% RSLogix 500 project TEST DENHAM_BAK006.RSS, saved by version 11.00.00.00 %
PROJECT "UNTITLED"    % processor: MicroLogix 1400 %

PROGRAM FILES
  LAD 2   184 rungs

DATA FILES
  O0 OUTPUT  8 elements
  I1 INPUT  17 elements
  S2 STATUS  66 elements
  B3 BINARY  6 elements
  T4 TIMER  28 elements
  C5 COUNTER  1 elements
  R6 CONTROL  1 elements
  N7 INTEGER  41 elements
  F8 FLOAT  8 elements
  PD11   2 elements

LADDER 2
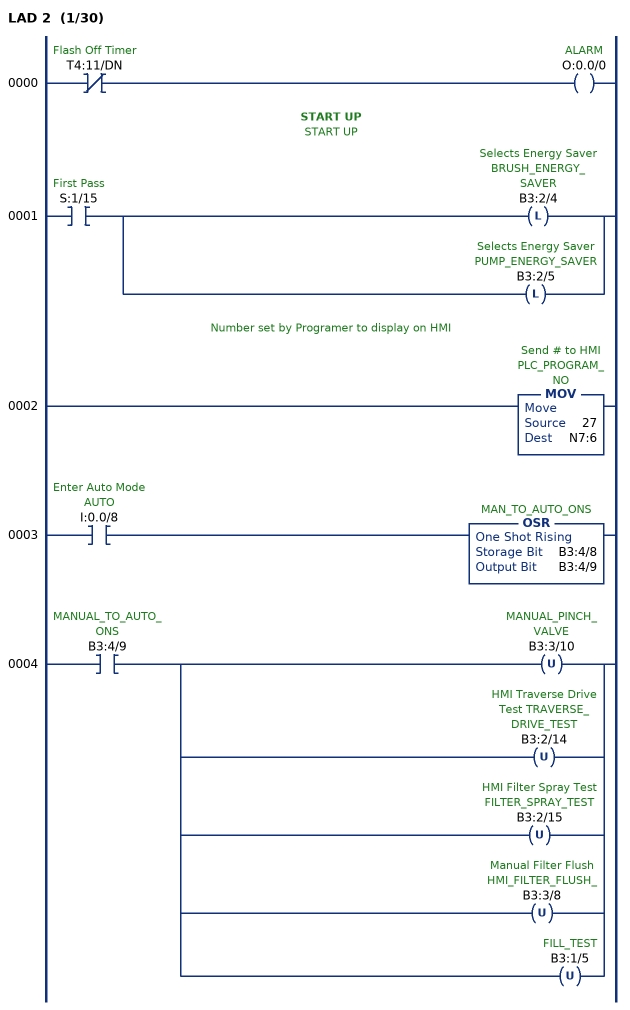
% Rung: 0 %
SOR XIO T4:11/DN OTE O:0.0/0 EOR
%   T4:11  "Flash Off Timer" %
%   O:0.0/0  ALARM %
% Rung: 1 %
% TITLE: START UP %
% START UP %
SOR XIC S:1/15 BST OTL B3:2/4 NXB OTL B3:2/5 BND EOR
%   S:1/15  "First Pass" %
%   B3:2/4  BRUSH_ENERGY_SAVER  "Selects Energy Saver" %
%   B3:2/5  PUMP_ENERGY_SAVER  "Selects Energy Saver" %
% Rung: 2 %
% Number set by Programer to display on HMI %
SOR MOV 27 N7:6 EOR
%   N7:6  PLC_PROGRAM_NO  "Send # to HMI" %
% Rung: 3 %
SOR XIC I:0.0/8 OSR B3:4/8 B3:4/9 EOR
%   I:0.0/8  AUTO  "Enter Auto Mode" %
%   B3:4/8  MAN_TO_AUTO_ONS %
%   B3:4/9  MANUAL_TO_AUTO_ONS %
% Rung: 4 %
SOR XIC B3:4/9 BST OTU B3:3/10 NXB BST OTU B3:2/14 NXB BST OTU B3:2/15 NXB BST OTU B3:3/8 NXB OTU B3:1/5 BND BND BND BND EOR
%   B3:4/9  MANUAL_TO_AUTO_ONS %
%   B3:3/10  MANUAL_PINCH_VALVE %
%   B3:2/14  TRAVERSE_DRIVE_TEST  "HMI Traverse Drive Test" %
%   B3:2/15  FILTER_SPRAY_TEST  "HMI Filter Spray Test" %
%   B3:3/8  HMI_FILTER_FLUSH_  "Manual Filter Flush" %
%   B3:1/5  FILL_TEST %

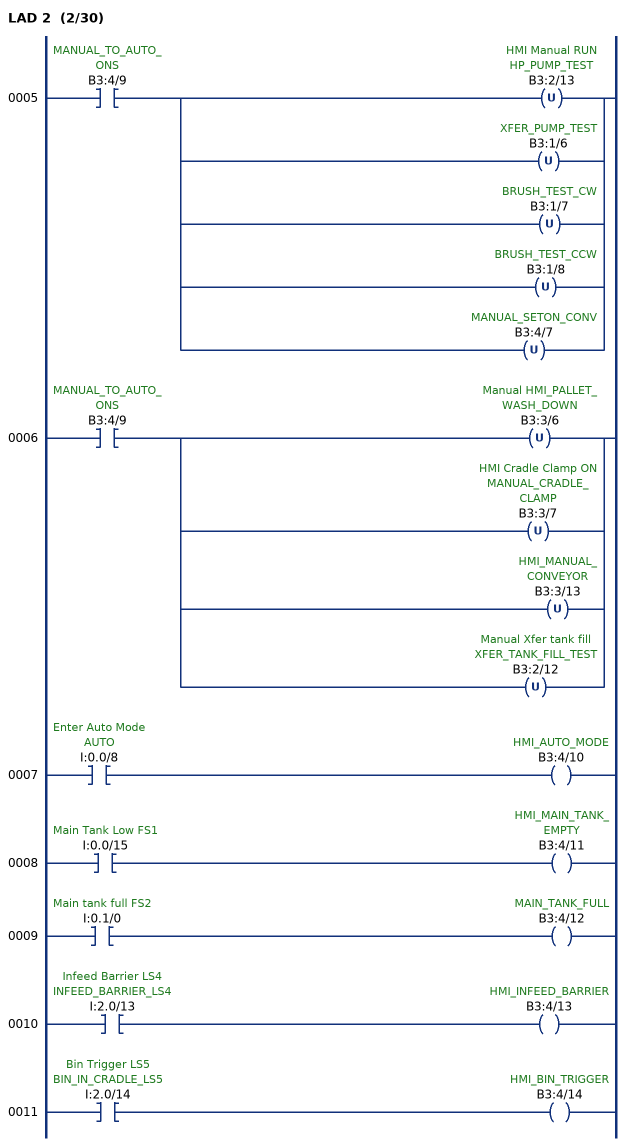
% Rung: 5 %
SOR XIC B3:4/9 BST OTU B3:2/13 NXB BST OTU B3:1/6 NXB BST OTU B3:1/7 NXB BST OTU B3:1/8 NXB OTU B3:4/7 BND BND BND BND EOR
%   B3:4/9  MANUAL_TO_AUTO_ONS %
%   B3:2/13  HP_PUMP_TEST  "HMI Manual RUN" %
%   B3:1/6  XFER_PUMP_TEST %
%   B3:1/7  BRUSH_TEST_CW %
%   B3:1/8  BRUSH_TEST_CCW %
%   B3:4/7  MANUAL_SETON_CONV %
% Rung: 6 %
SOR XIC B3:4/9 BST OTU B3:3/6 NXB BST OTU B3:3/7 NXB BST OTU B3:3/13 NXB OTU B3:2/12 BND BND BND EOR
%   B3:4/9  MANUAL_TO_AUTO_ONS %
%   B3:3/6  HMI_PALLET_WASH_DOWN  "Manual" %
%   B3:3/7  MANUAL_CRADLE_CLAMP  "HMI Cradle Clamp ON" %
%   B3:3/13  HMI_MANUAL_CONVEYOR %
%   B3:2/12  XFER_TANK_FILL_TEST  "Manual Xfer tank fill" %
% Rung: 7 %
SOR XIC I:0.0/8 OTE B3:4/10 EOR
%   I:0.0/8  AUTO  "Enter Auto Mode" %
%   B3:4/10  HMI_AUTO_MODE %
% Rung: 8 %
SOR XIC I:0.0/15 OTE B3:4/11 EOR
%   I:0.0/15  FS1  "Main Tank Low" %
%   B3:4/11  HMI_MAIN_TANK_EMPTY %
% Rung: 9 %
SOR XIC I:0.1/0 OTE B3:4/12 EOR
%   I:0.1/0  FS2  "Main tank full" %
%   B3:4/12  MAIN_TANK_FULL %
% Rung: 10 %
SOR XIC I:2.0/13 OTE B3:4/13 EOR
%   I:2.0/13  INFEED_BARRIER_LS4  "Infeed Barrier LS4" %
%   B3:4/13  HMI_INFEED_BARRIER %
% Rung: 11 %
SOR XIC I:2.0/14 OTE B3:4/14 EOR
%   I:2.0/14  BIN_IN_CRADLE_LS5  "Bin Trigger LS5" %
%   B3:4/14  HMI_BIN_TRIGGER %

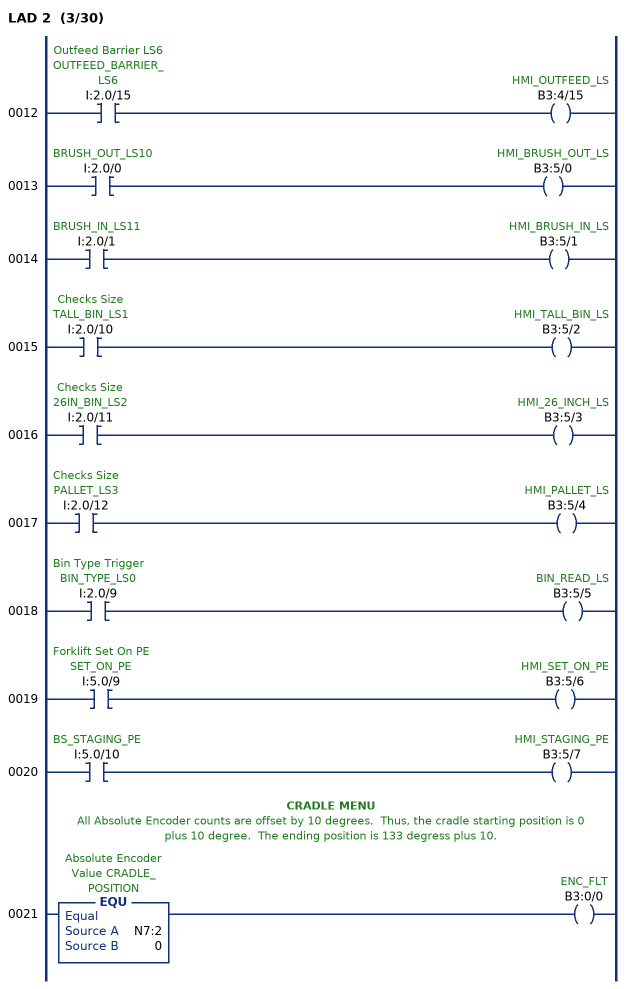
% Rung: 12 %
SOR XIC I:2.0/15 OTE B3:4/15 EOR
%   I:2.0/15  OUTFEED_BARRIER_LS6  "Outfeed Barrier LS6" %
%   B3:4/15  HMI_OUTFEED_LS %
% Rung: 13 %
SOR XIC I:2.0/0 OTE B3:5/0 EOR
%   I:2.0/0  BRUSH_OUT_LS10 %
%   B3:5/0  HMI_BRUSH_OUT_LS %
% Rung: 14 %
SOR XIC I:2.0/1 OTE B3:5/1 EOR
%   I:2.0/1  BRUSH_IN_LS11 %
%   B3:5/1  HMI_BRUSH_IN_LS %
% Rung: 15 %
SOR XIC I:2.0/10 OTE B3:5/2 EOR
%   I:2.0/10  TALL_BIN_LS1  "Checks Size" %
%   B3:5/2  HMI_TALL_BIN_LS %
% Rung: 16 %
SOR XIC I:2.0/11 OTE B3:5/3 EOR
%   I:2.0/11  26IN_BIN_LS2  "Checks Size" %
%   B3:5/3  HMI_26_INCH_LS %
% Rung: 17 %
SOR XIC I:2.0/12 OTE B3:5/4 EOR
%   I:2.0/12  PALLET_LS3  "Checks Size" %
%   B3:5/4  HMI_PALLET_LS %
% Rung: 18 %
SOR XIC I:2.0/9 OTE B3:5/5 EOR
%   I:2.0/9  BIN_TYPE_LS0  "Bin Type Trigger" %
%   B3:5/5  BIN_READ_LS %
% Rung: 19 %
SOR XIC I:5.0/9 OTE B3:5/6 EOR
%   I:5.0/9  SET_ON_PE  "Forklift Set On PE" %
%   B3:5/6  HMI_SET_ON_PE %
% Rung: 20 %
SOR XIC I:5.0/10 OTE B3:5/7 EOR
%   I:5.0/10  BS_STAGING_PE %
%   B3:5/7  HMI_STAGING_PE %
% Rung: 21 %
% TITLE: CRADLE MENU %
% All Absolute Encoder counts are offset by 10 degrees.  Thus, the cradle starting position is 0 plus 10 degree.  The ending position is 133 degress plus 10. %
SOR EQU N7:2 0 OTE B3:0/0 EOR
%   N7:2  CRADLE_POSITION  "Absolute Encoder Value" %
%   B3:0/0  ENC_FLT %

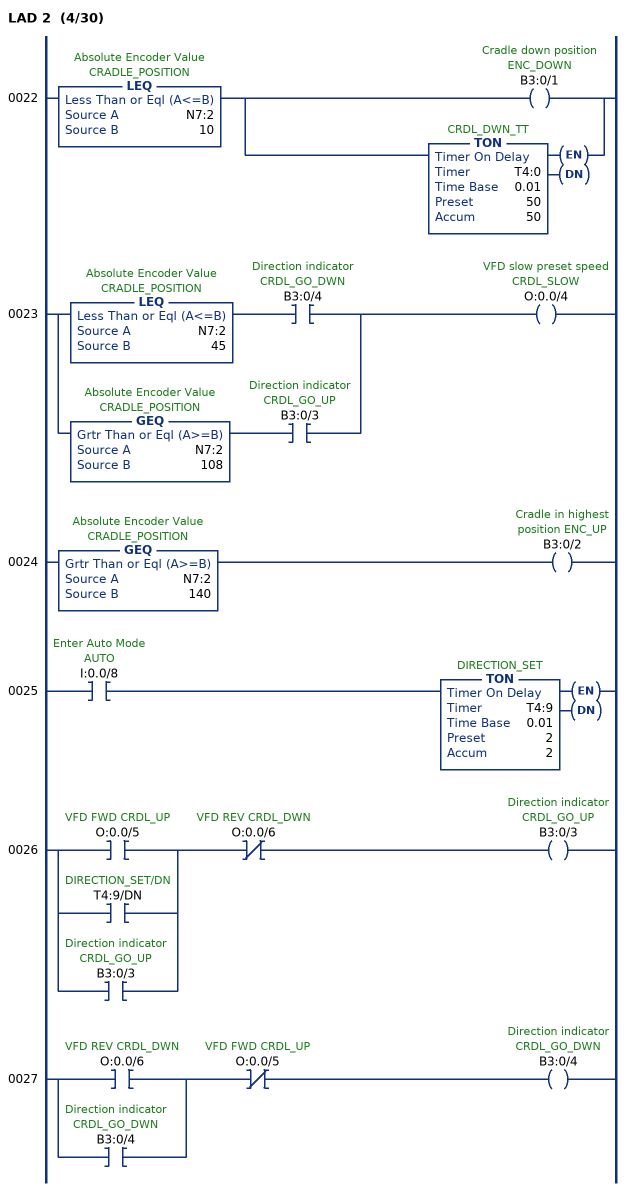
% Rung: 22 %
SOR LEQ N7:2 10 BST OTE B3:0/1 NXB TON T4:0 0.01 50 50 BND EOR
%   N7:2  CRADLE_POSITION  "Absolute Encoder Value" %
%   B3:0/1  ENC_DOWN  "Cradle down position" %
%   T4:0  CRDL_DWN_TT %
% Rung: 23 %
SOR BST LEQ N7:2 45 XIC B3:0/4 NXB GEQ N7:2 108 XIC B3:0/3 BND OTE O:0.0/4 EOR
%   N7:2  CRADLE_POSITION  "Absolute Encoder Value" %
%   B3:0/4  CRDL_GO_DWN  "Direction indicator" %
%   B3:0/3  CRDL_GO_UP  "Direction indicator" %
%   O:0.0/4  CRDL_SLOW  "VFD slow preset speed" %
% Rung: 24 %
SOR GEQ N7:2 140 OTE B3:0/2 EOR
%   N7:2  CRADLE_POSITION  "Absolute Encoder Value" %
%   B3:0/2  ENC_UP  "Cradle in highest position" %
% Rung: 25 %
SOR XIC I:0.0/8 TON T4:9 0.01 2 2 EOR
%   I:0.0/8  AUTO  "Enter Auto Mode" %
%   T4:9  DIRECTION_SET %
% Rung: 26 %
SOR BST XIC O:0.0/5 NXB XIC T4:9/DN NXB XIC B3:0/3 BND XIO O:0.0/6 OTE B3:0/3 EOR
%   O:0.0/5  CRDL_UP  "VFD FWD" %
%   T4:9  DIRECTION_SET %
%   B3:0/3  CRDL_GO_UP  "Direction indicator" %
%   O:0.0/6  CRDL_DWN  "VFD REV" %
% Rung: 27 %
SOR BST XIC O:0.0/6 NXB XIC B3:0/4 BND XIO O:0.0/5 OTE B3:0/4 EOR
%   O:0.0/6  CRDL_DWN  "VFD REV" %
%   B3:0/4  CRDL_GO_DWN  "Direction indicator" %
%   O:0.0/5  CRDL_UP  "VFD FWD" %

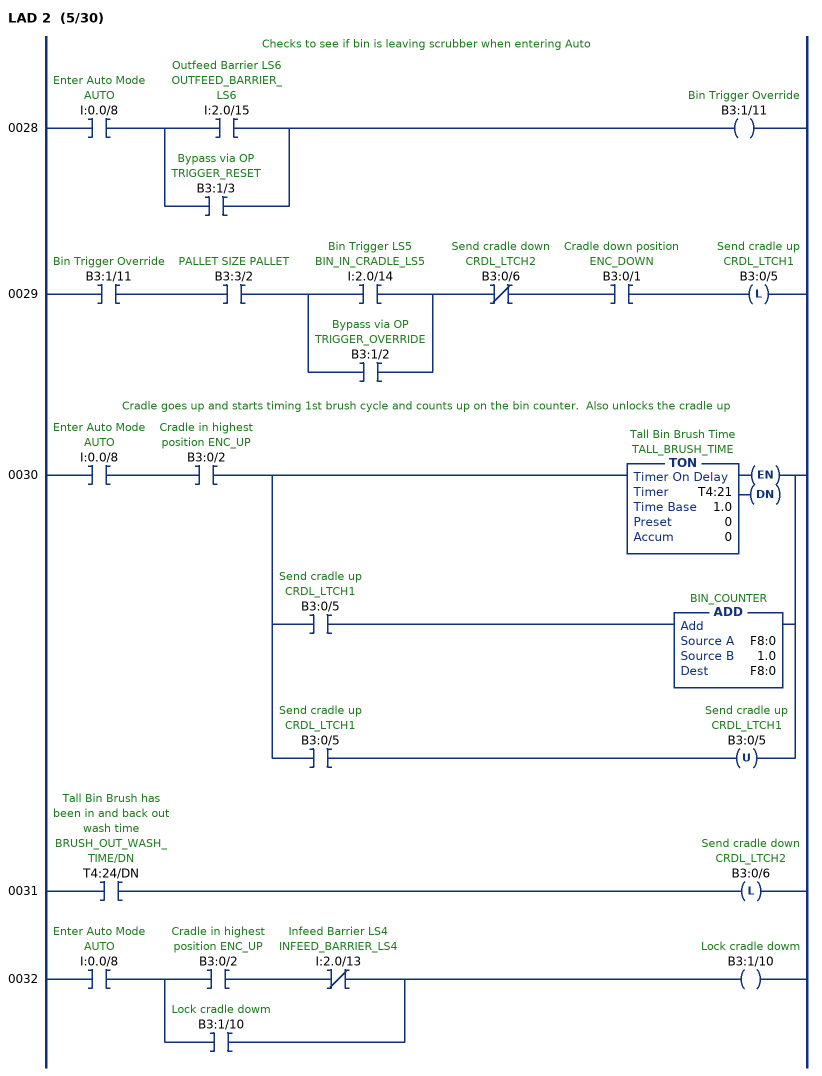
% Rung: 28 %
% Checks to see if bin is leaving scrubber when entering Auto %
SOR XIC I:0.0/8 BST XIC I:2.0/15 NXB XIC B3:1/3 BND OTE B3:1/11 EOR
%   I:0.0/8  AUTO  "Enter Auto Mode" %
%   I:2.0/15  OUTFEED_BARRIER_LS6  "Outfeed Barrier LS6" %
%   B3:1/3  TRIGGER_RESET  "Bypass via OP" %
%   B3:1/11  "Bin Trigger Override" %
% Rung: 29 %
SOR XIC B3:1/11 XIC B3:3/2 BST XIC I:2.0/14 NXB XIC B3:1/2 BND XIO B3:0/6 XIC B3:0/1 OTL B3:0/5 EOR
%   B3:1/11  "Bin Trigger Override" %
%   B3:3/2  PALLET  "PALLET SIZE" %
%   I:2.0/14  BIN_IN_CRADLE_LS5  "Bin Trigger LS5" %
%   B3:1/2  TRIGGER_OVERRIDE  "Bypass via OP" %
%   B3:0/6  CRDL_LTCH2  "Send cradle down" %
%   B3:0/1  ENC_DOWN  "Cradle down position" %
%   B3:0/5  CRDL_LTCH1  "Send cradle up" %
% Rung: 30 %
% Cradle goes up and starts timing 1st brush cycle and counts up on the bin counter.  Also unlocks the cradle up %
SOR XIC I:0.0/8 XIC B3:0/2 BST TON T4:21 1.0 0 0 NXB BST XIC B3:0/5 ADD F8:0 1.0 F8:0 NXB XIC B3:0/5 OTU B3:0/5 BND BND EOR
%   I:0.0/8  AUTO  "Enter Auto Mode" %
%   B3:0/2  ENC_UP  "Cradle in highest position" %
%   T4:21  TALL_BRUSH_TIME  "Tall Bin Brush Time" %
%   B3:0/5  CRDL_LTCH1  "Send cradle up" %
%   F8:0  BIN_COUNTER %
% Rung: 31 %
SOR XIC T4:24/DN OTL B3:0/6 EOR
%   T4:24  BRUSH_OUT_WASH_TIME  "Tall Bin Brush has been in and back out wash time" %
%   B3:0/6  CRDL_LTCH2  "Send cradle down" %
% Rung: 32 %
SOR XIC I:0.0/8 BST XIC B3:0/2 XIO I:2.0/13 NXB XIC B3:1/10 BND OTE B3:1/10 EOR
%   I:0.0/8  AUTO  "Enter Auto Mode" %
%   B3:0/2  ENC_UP  "Cradle in highest position" %
%   I:2.0/13  INFEED_BARRIER_LS4  "Infeed Barrier LS4" %
%   B3:1/10  "Lock cradle dowm" %

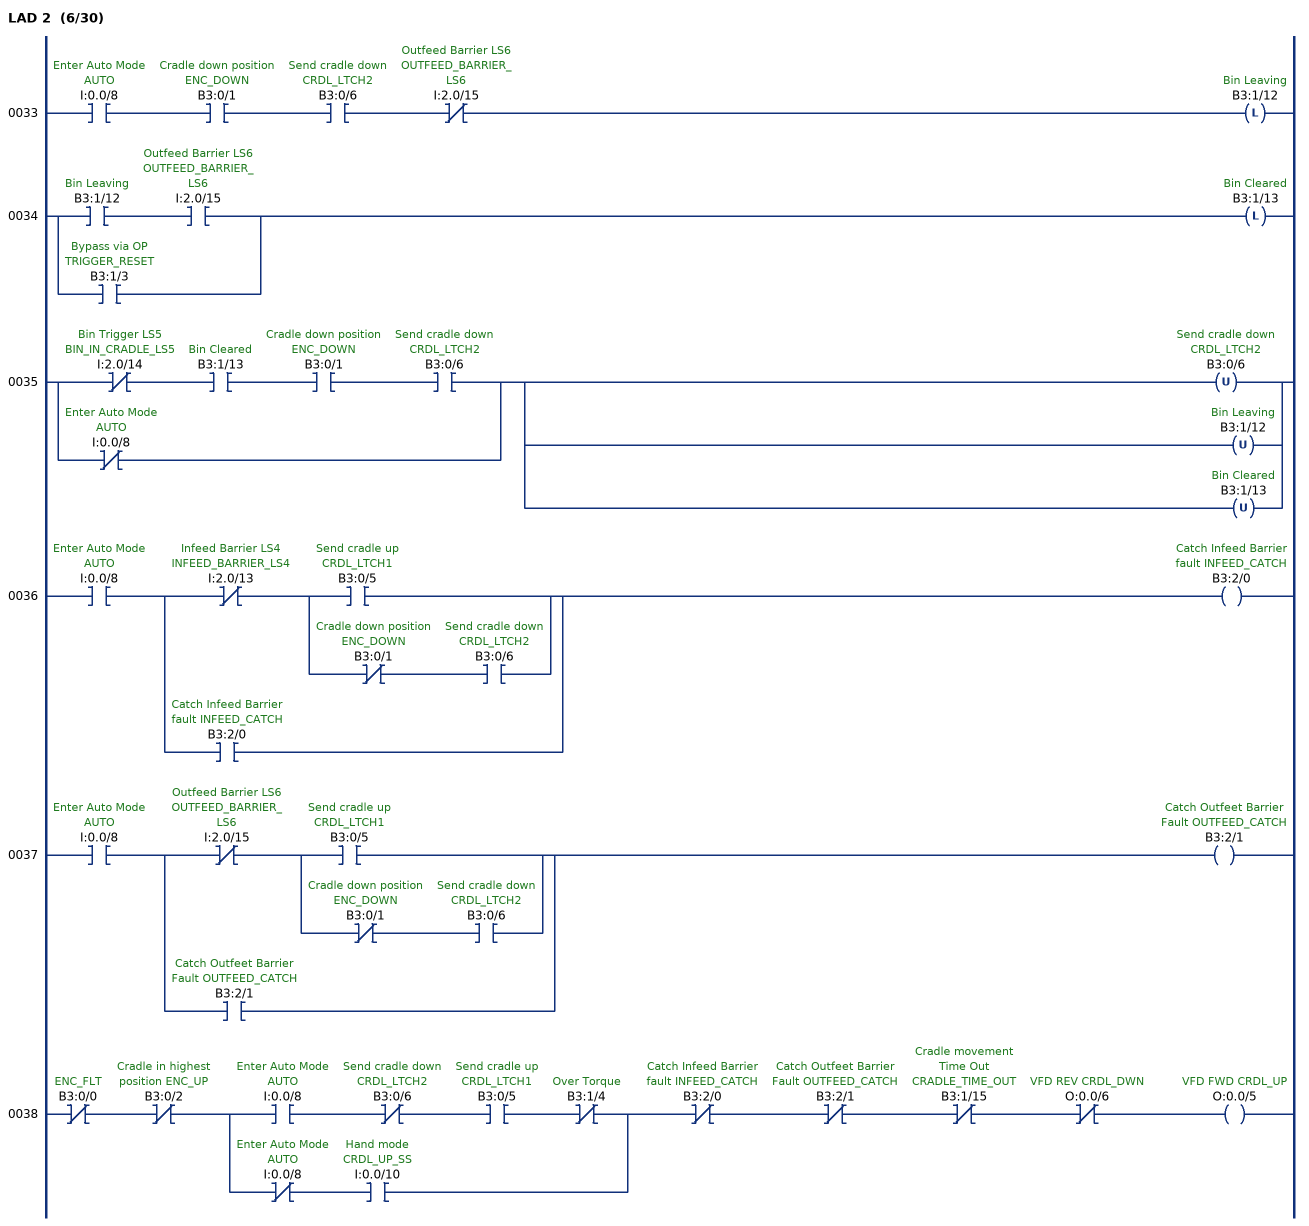
% Rung: 33 %
SOR XIC I:0.0/8 XIC B3:0/1 XIC B3:0/6 XIO I:2.0/15 OTL B3:1/12 EOR
%   I:0.0/8  AUTO  "Enter Auto Mode" %
%   B3:0/1  ENC_DOWN  "Cradle down position" %
%   B3:0/6  CRDL_LTCH2  "Send cradle down" %
%   I:2.0/15  OUTFEED_BARRIER_LS6  "Outfeed Barrier LS6" %
%   B3:1/12  "Bin Leaving" %
% Rung: 34 %
SOR BST XIC B3:1/12 XIC I:2.0/15 NXB XIC B3:1/3 BND OTL B3:1/13 EOR
%   B3:1/12  "Bin Leaving" %
%   I:2.0/15  OUTFEED_BARRIER_LS6  "Outfeed Barrier LS6" %
%   B3:1/3  TRIGGER_RESET  "Bypass via OP" %
%   B3:1/13  "Bin Cleared" %
% Rung: 35 %
SOR BST XIO I:2.0/14 XIC B3:1/13 XIC B3:0/1 XIC B3:0/6 NXB XIO I:0.0/8 BND BST OTU B3:0/6 NXB BST OTU B3:1/12 NXB OTU B3:1/13 BND BND EOR
%   I:2.0/14  BIN_IN_CRADLE_LS5  "Bin Trigger LS5" %
%   B3:1/13  "Bin Cleared" %
%   B3:0/1  ENC_DOWN  "Cradle down position" %
%   B3:0/6  CRDL_LTCH2  "Send cradle down" %
%   I:0.0/8  AUTO  "Enter Auto Mode" %
%   B3:1/12  "Bin Leaving" %
% Rung: 36 %
SOR XIC I:0.0/8 BST XIO I:2.0/13 BST XIC B3:0/5 NXB XIO B3:0/1 XIC B3:0/6 BND NXB XIC B3:2/0 BND OTE B3:2/0 EOR
%   I:0.0/8  AUTO  "Enter Auto Mode" %
%   I:2.0/13  INFEED_BARRIER_LS4  "Infeed Barrier LS4" %
%   B3:0/5  CRDL_LTCH1  "Send cradle up" %
%   B3:0/1  ENC_DOWN  "Cradle down position" %
%   B3:0/6  CRDL_LTCH2  "Send cradle down" %
%   B3:2/0  INFEED_CATCH  "Catch Infeed Barrier fault" %
% Rung: 37 %
SOR XIC I:0.0/8 BST XIO I:2.0/15 BST XIC B3:0/5 NXB XIO B3:0/1 XIC B3:0/6 BND NXB XIC B3:2/1 BND OTE B3:2/1 EOR
%   I:0.0/8  AUTO  "Enter Auto Mode" %
%   I:2.0/15  OUTFEED_BARRIER_LS6  "Outfeed Barrier LS6" %
%   B3:0/5  CRDL_LTCH1  "Send cradle up" %
%   B3:0/1  ENC_DOWN  "Cradle down position" %
%   B3:0/6  CRDL_LTCH2  "Send cradle down" %
%   B3:2/1  OUTFEED_CATCH  "Catch Outfeet Barrier Fault" %
% Rung: 38 %
SOR XIO B3:0/0 XIO B3:0/2 BST XIC I:0.0/8 XIO B3:0/6 XIC B3:0/5 XIO B3:1/4 NXB XIO I:0.0/8 XIC I:0.0/10 BND XIO B3:2/0 XIO B3:2/1 XIO B3:1/15 XIO O:0.0/6 OTE O:0.0/5 EOR
%   B3:0/0  ENC_FLT %
%   B3:0/2  ENC_UP  "Cradle in highest position" %
%   I:0.0/8  AUTO  "Enter Auto Mode" %
%   B3:0/6  CRDL_LTCH2  "Send cradle down" %
%   B3:0/5  CRDL_LTCH1  "Send cradle up" %
%   B3:1/4  "Over Torque" %
%   I:0.0/10  CRDL_UP_SS  "Hand mode" %
%   B3:2/0  INFEED_CATCH  "Catch Infeed Barrier fault" %
%   B3:2/1  OUTFEED_CATCH  "Catch Outfeet Barrier Fault" %
%   B3:1/15  CRADLE_TIME_OUT  "Cradle movement Time Out" %
%   O:0.0/6  CRDL_DWN  "VFD REV" %
%   O:0.0/5  CRDL_UP  "VFD FWD" %

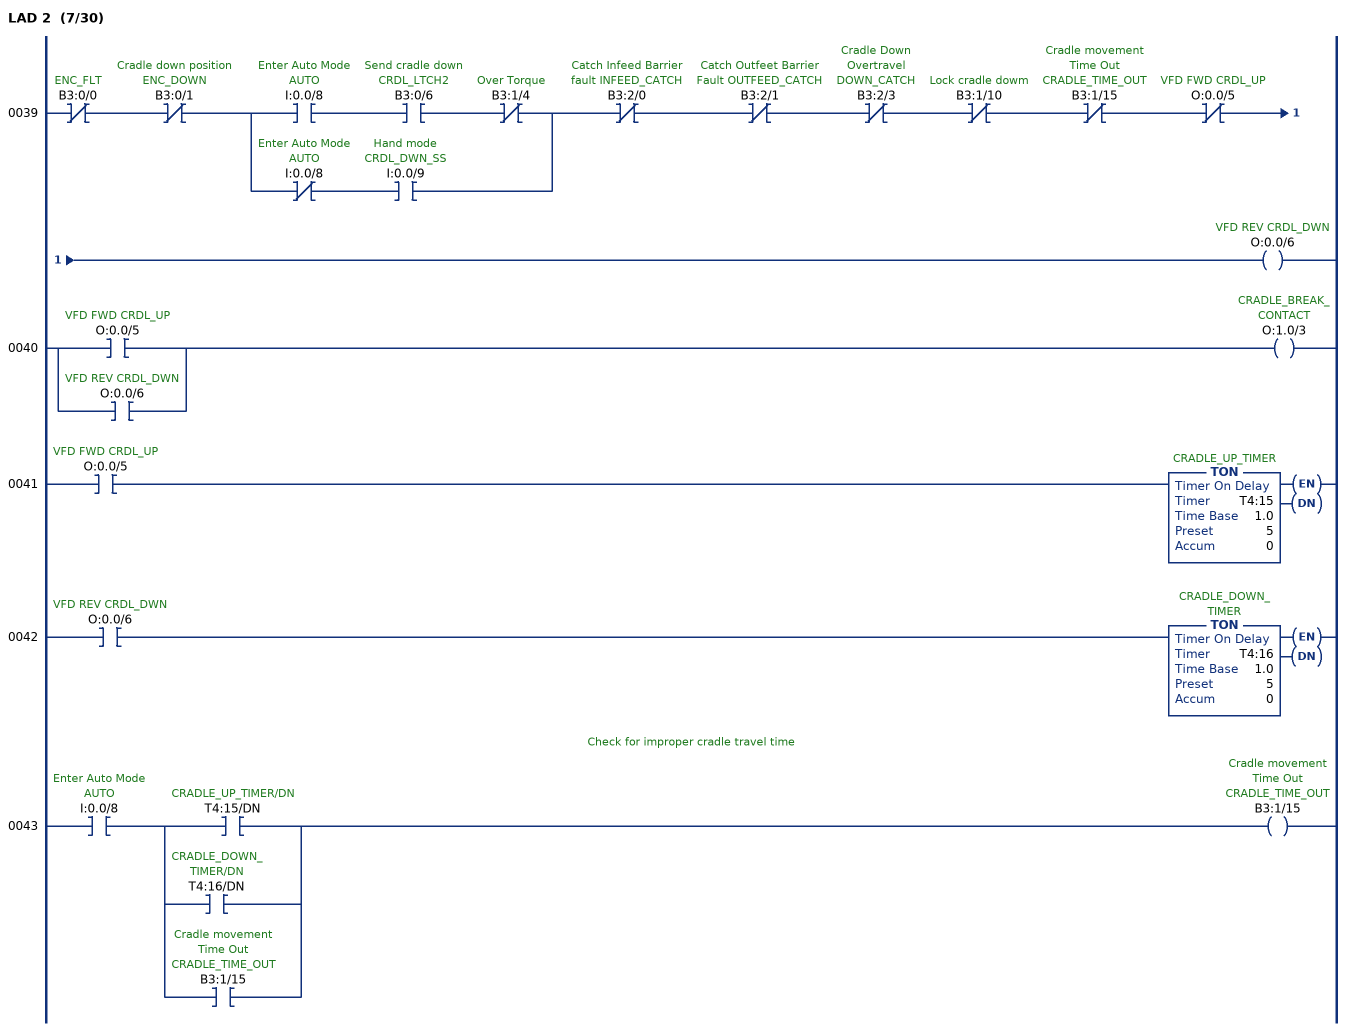
% Rung: 39 %
SOR XIO B3:0/0 XIO B3:0/1 BST XIC I:0.0/8 XIC B3:0/6 XIO B3:1/4 NXB XIO I:0.0/8 XIC I:0.0/9 BND XIO B3:2/0 XIO B3:2/1 XIO B3:2/3 XIO B3:1/10 XIO B3:1/15 XIO O:0.0/5 OTE O:0.0/6 EOR
%   B3:0/0  ENC_FLT %
%   B3:0/1  ENC_DOWN  "Cradle down position" %
%   I:0.0/8  AUTO  "Enter Auto Mode" %
%   B3:0/6  CRDL_LTCH2  "Send cradle down" %
%   B3:1/4  "Over Torque" %
%   I:0.0/9  CRDL_DWN_SS  "Hand mode" %
%   B3:2/0  INFEED_CATCH  "Catch Infeed Barrier fault" %
%   B3:2/1  OUTFEED_CATCH  "Catch Outfeet Barrier Fault" %
%   B3:2/3  DOWN_CATCH  "Cradle Down Overtravel" %
%   B3:1/10  "Lock cradle dowm" %
%   B3:1/15  CRADLE_TIME_OUT  "Cradle movement Time Out" %
%   O:0.0/5  CRDL_UP  "VFD FWD" %
%   O:0.0/6  CRDL_DWN  "VFD REV" %
% Rung: 40 %
SOR BST XIC O:0.0/5 NXB XIC O:0.0/6 BND OTE O:1.0/3 EOR
%   O:0.0/5  CRDL_UP  "VFD FWD" %
%   O:0.0/6  CRDL_DWN  "VFD REV" %
%   O:1.0/3  CRADLE_BREAK_CONTACT %
% Rung: 41 %
SOR XIC O:0.0/5 TON T4:15 1.0 5 0 EOR
%   O:0.0/5  CRDL_UP  "VFD FWD" %
%   T4:15  CRADLE_UP_TIMER %
% Rung: 42 %
SOR XIC O:0.0/6 TON T4:16 1.0 5 0 EOR
%   O:0.0/6  CRDL_DWN  "VFD REV" %
%   T4:16  CRADLE_DOWN_TIMER %
% Rung: 43 %
% Check for improper cradle travel time %
SOR XIC I:0.0/8 BST BST XIC T4:15/DN NXB XIC T4:16/DN BND NXB XIC B3:1/15 BND OTE B3:1/15 EOR
%   I:0.0/8  AUTO  "Enter Auto Mode" %
%   T4:15  CRADLE_UP_TIMER %
%   T4:16  CRADLE_DOWN_TIMER %
%   B3:1/15  CRADLE_TIME_OUT  "Cradle movement Time Out" %

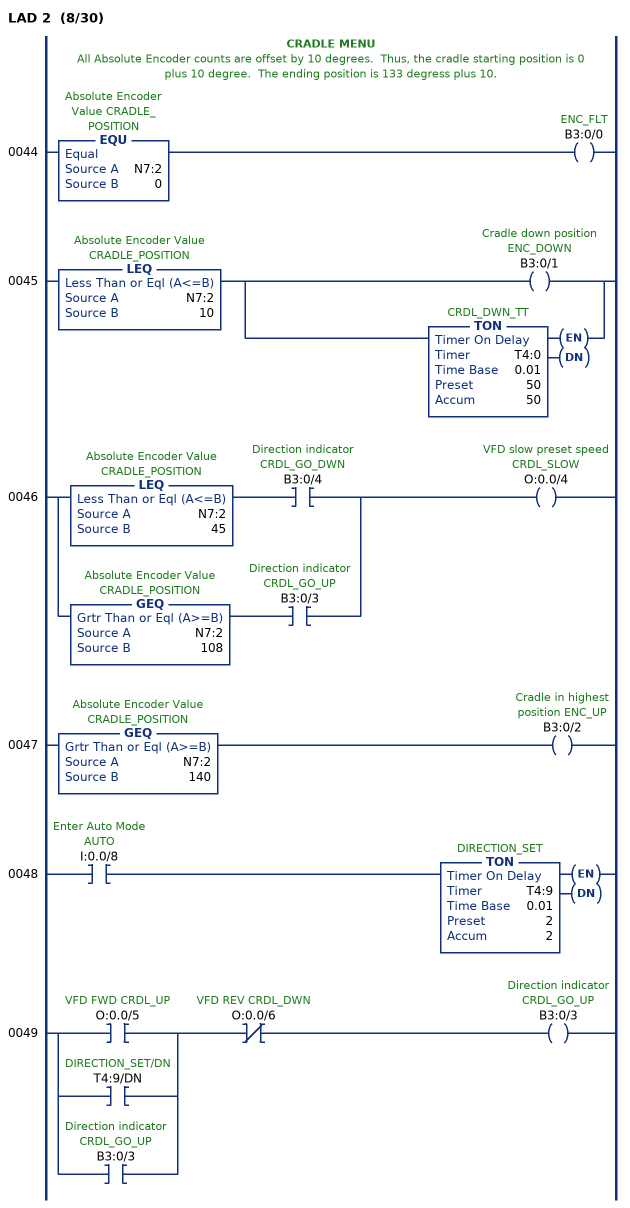
% Rung: 44 %
% TITLE: CRADLE MENU %
% All Absolute Encoder counts are offset by 10 degrees.  Thus, the cradle starting position is 0 plus 10 degree.  The ending position is 133 degress plus 10. %
SOR EQU N7:2 0 OTE B3:0/0 EOR
%   N7:2  CRADLE_POSITION  "Absolute Encoder Value" %
%   B3:0/0  ENC_FLT %
% Rung: 45 %
SOR LEQ N7:2 10 BST OTE B3:0/1 NXB TON T4:0 0.01 50 50 BND EOR
%   N7:2  CRADLE_POSITION  "Absolute Encoder Value" %
%   B3:0/1  ENC_DOWN  "Cradle down position" %
%   T4:0  CRDL_DWN_TT %
% Rung: 46 %
SOR BST LEQ N7:2 45 XIC B3:0/4 NXB GEQ N7:2 108 XIC B3:0/3 BND OTE O:0.0/4 EOR
%   N7:2  CRADLE_POSITION  "Absolute Encoder Value" %
%   B3:0/4  CRDL_GO_DWN  "Direction indicator" %
%   B3:0/3  CRDL_GO_UP  "Direction indicator" %
%   O:0.0/4  CRDL_SLOW  "VFD slow preset speed" %
% Rung: 47 %
SOR GEQ N7:2 140 OTE B3:0/2 EOR
%   N7:2  CRADLE_POSITION  "Absolute Encoder Value" %
%   B3:0/2  ENC_UP  "Cradle in highest position" %
% Rung: 48 %
SOR XIC I:0.0/8 TON T4:9 0.01 2 2 EOR
%   I:0.0/8  AUTO  "Enter Auto Mode" %
%   T4:9  DIRECTION_SET %
% Rung: 49 %
SOR BST XIC O:0.0/5 NXB XIC T4:9/DN NXB XIC B3:0/3 BND XIO O:0.0/6 OTE B3:0/3 EOR
%   O:0.0/5  CRDL_UP  "VFD FWD" %
%   T4:9  DIRECTION_SET %
%   B3:0/3  CRDL_GO_UP  "Direction indicator" %
%   O:0.0/6  CRDL_DWN  "VFD REV" %

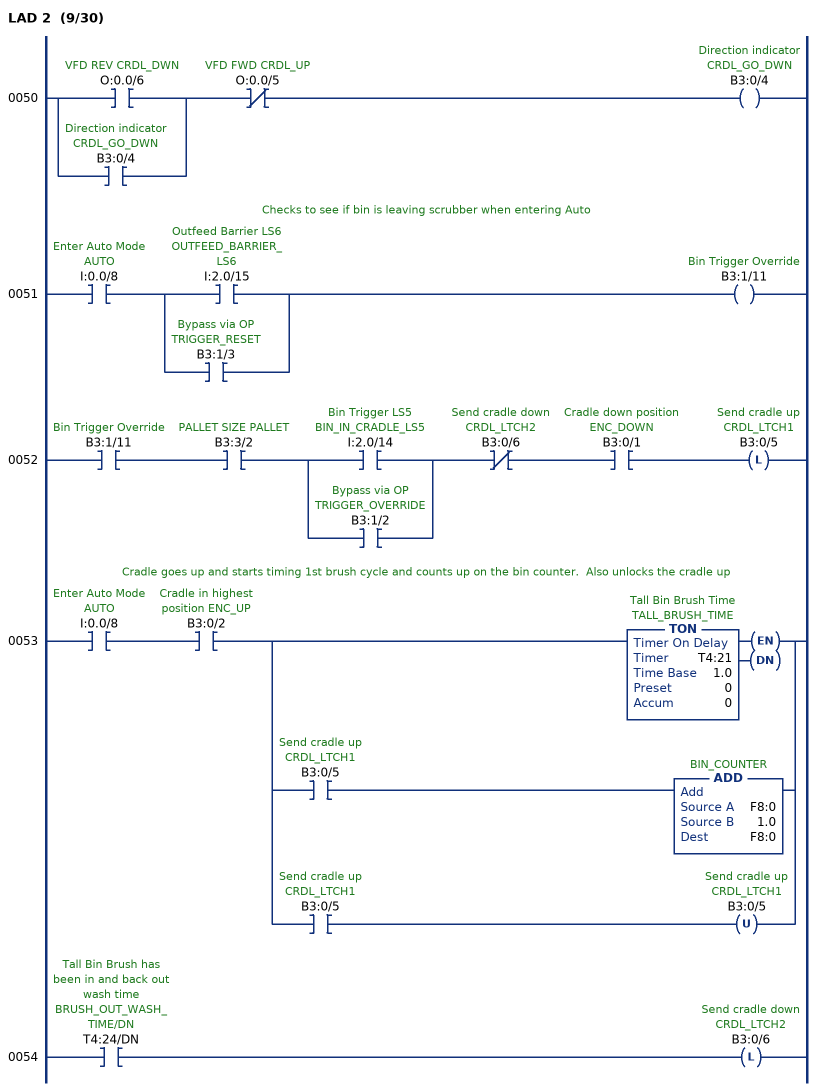
% Rung: 50 %
SOR BST XIC O:0.0/6 NXB XIC B3:0/4 BND XIO O:0.0/5 OTE B3:0/4 EOR
%   O:0.0/6  CRDL_DWN  "VFD REV" %
%   B3:0/4  CRDL_GO_DWN  "Direction indicator" %
%   O:0.0/5  CRDL_UP  "VFD FWD" %
% Rung: 51 %
% Checks to see if bin is leaving scrubber when entering Auto %
SOR XIC I:0.0/8 BST XIC I:2.0/15 NXB XIC B3:1/3 BND OTE B3:1/11 EOR
%   I:0.0/8  AUTO  "Enter Auto Mode" %
%   I:2.0/15  OUTFEED_BARRIER_LS6  "Outfeed Barrier LS6" %
%   B3:1/3  TRIGGER_RESET  "Bypass via OP" %
%   B3:1/11  "Bin Trigger Override" %
% Rung: 52 %
SOR XIC B3:1/11 XIC B3:3/2 BST XIC I:2.0/14 NXB XIC B3:1/2 BND XIO B3:0/6 XIC B3:0/1 OTL B3:0/5 EOR
%   B3:1/11  "Bin Trigger Override" %
%   B3:3/2  PALLET  "PALLET SIZE" %
%   I:2.0/14  BIN_IN_CRADLE_LS5  "Bin Trigger LS5" %
%   B3:1/2  TRIGGER_OVERRIDE  "Bypass via OP" %
%   B3:0/6  CRDL_LTCH2  "Send cradle down" %
%   B3:0/1  ENC_DOWN  "Cradle down position" %
%   B3:0/5  CRDL_LTCH1  "Send cradle up" %
% Rung: 53 %
% Cradle goes up and starts timing 1st brush cycle and counts up on the bin counter.  Also unlocks the cradle up %
SOR XIC I:0.0/8 XIC B3:0/2 BST TON T4:21 1.0 0 0 NXB BST XIC B3:0/5 ADD F8:0 1.0 F8:0 NXB XIC B3:0/5 OTU B3:0/5 BND BND EOR
%   I:0.0/8  AUTO  "Enter Auto Mode" %
%   B3:0/2  ENC_UP  "Cradle in highest position" %
%   T4:21  TALL_BRUSH_TIME  "Tall Bin Brush Time" %
%   B3:0/5  CRDL_LTCH1  "Send cradle up" %
%   F8:0  BIN_COUNTER %
% Rung: 54 %
SOR XIC T4:24/DN OTL B3:0/6 EOR
%   T4:24  BRUSH_OUT_WASH_TIME  "Tall Bin Brush has been in and back out wash time" %
%   B3:0/6  CRDL_LTCH2  "Send cradle down" %

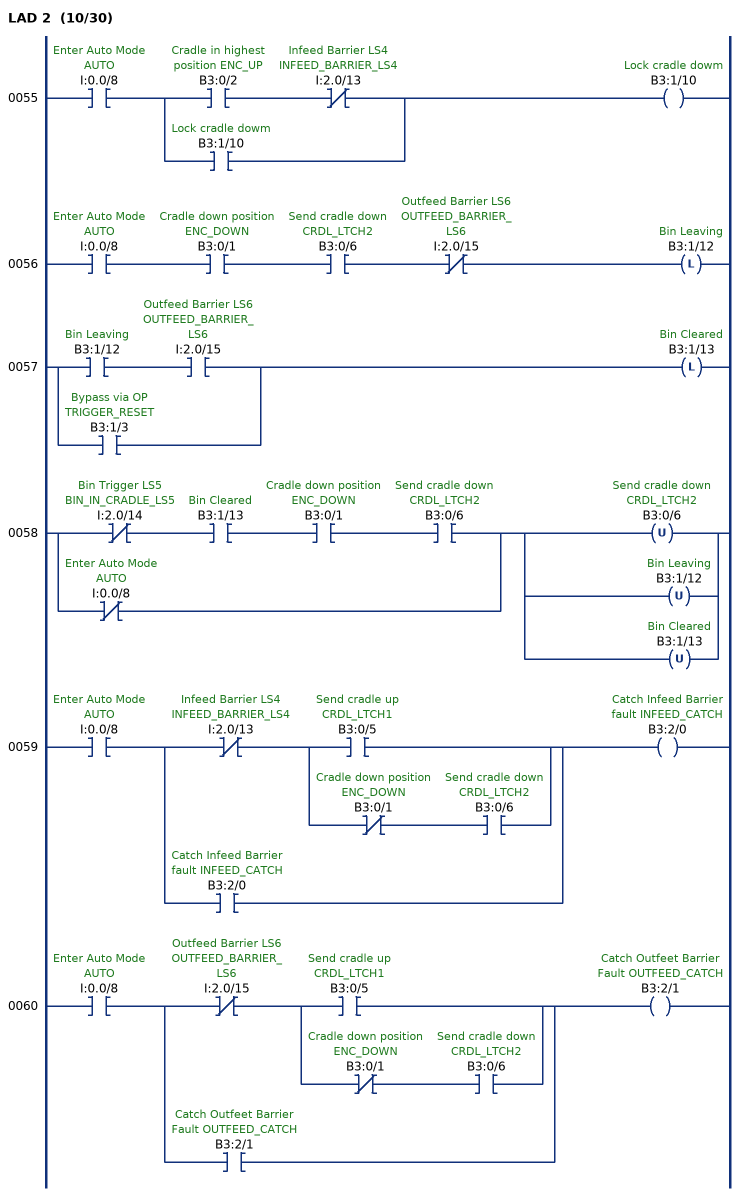
% Rung: 55 %
SOR XIC I:0.0/8 BST XIC B3:0/2 XIO I:2.0/13 NXB XIC B3:1/10 BND OTE B3:1/10 EOR
%   I:0.0/8  AUTO  "Enter Auto Mode" %
%   B3:0/2  ENC_UP  "Cradle in highest position" %
%   I:2.0/13  INFEED_BARRIER_LS4  "Infeed Barrier LS4" %
%   B3:1/10  "Lock cradle dowm" %
% Rung: 56 %
SOR XIC I:0.0/8 XIC B3:0/1 XIC B3:0/6 XIO I:2.0/15 OTL B3:1/12 EOR
%   I:0.0/8  AUTO  "Enter Auto Mode" %
%   B3:0/1  ENC_DOWN  "Cradle down position" %
%   B3:0/6  CRDL_LTCH2  "Send cradle down" %
%   I:2.0/15  OUTFEED_BARRIER_LS6  "Outfeed Barrier LS6" %
%   B3:1/12  "Bin Leaving" %
% Rung: 57 %
SOR BST XIC B3:1/12 XIC I:2.0/15 NXB XIC B3:1/3 BND OTL B3:1/13 EOR
%   B3:1/12  "Bin Leaving" %
%   I:2.0/15  OUTFEED_BARRIER_LS6  "Outfeed Barrier LS6" %
%   B3:1/3  TRIGGER_RESET  "Bypass via OP" %
%   B3:1/13  "Bin Cleared" %
% Rung: 58 %
SOR BST XIO I:2.0/14 XIC B3:1/13 XIC B3:0/1 XIC B3:0/6 NXB XIO I:0.0/8 BND BST OTU B3:0/6 NXB BST OTU B3:1/12 NXB OTU B3:1/13 BND BND EOR
%   I:2.0/14  BIN_IN_CRADLE_LS5  "Bin Trigger LS5" %
%   B3:1/13  "Bin Cleared" %
%   B3:0/1  ENC_DOWN  "Cradle down position" %
%   B3:0/6  CRDL_LTCH2  "Send cradle down" %
%   I:0.0/8  AUTO  "Enter Auto Mode" %
%   B3:1/12  "Bin Leaving" %
% Rung: 59 %
SOR XIC I:0.0/8 BST XIO I:2.0/13 BST XIC B3:0/5 NXB XIO B3:0/1 XIC B3:0/6 BND NXB XIC B3:2/0 BND OTE B3:2/0 EOR
%   I:0.0/8  AUTO  "Enter Auto Mode" %
%   I:2.0/13  INFEED_BARRIER_LS4  "Infeed Barrier LS4" %
%   B3:0/5  CRDL_LTCH1  "Send cradle up" %
%   B3:0/1  ENC_DOWN  "Cradle down position" %
%   B3:0/6  CRDL_LTCH2  "Send cradle down" %
%   B3:2/0  INFEED_CATCH  "Catch Infeed Barrier fault" %
% Rung: 60 %
SOR XIC I:0.0/8 BST XIO I:2.0/15 BST XIC B3:0/5 NXB XIO B3:0/1 XIC B3:0/6 BND NXB XIC B3:2/1 BND OTE B3:2/1 EOR
%   I:0.0/8  AUTO  "Enter Auto Mode" %
%   I:2.0/15  OUTFEED_BARRIER_LS6  "Outfeed Barrier LS6" %
%   B3:0/5  CRDL_LTCH1  "Send cradle up" %
%   B3:0/1  ENC_DOWN  "Cradle down position" %
%   B3:0/6  CRDL_LTCH2  "Send cradle down" %
%   B3:2/1  OUTFEED_CATCH  "Catch Outfeet Barrier Fault" %

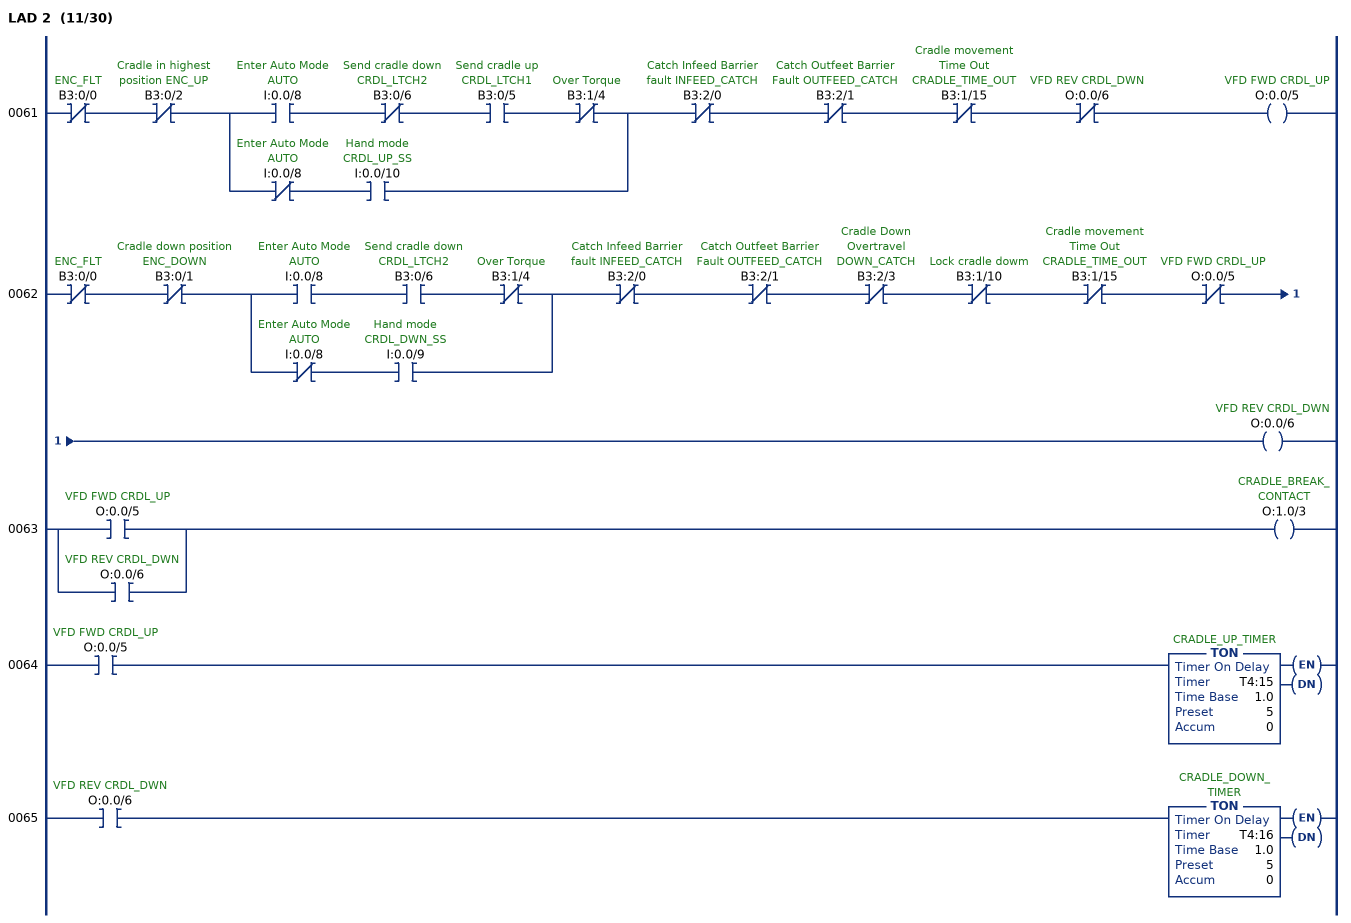
% Rung: 61 %
SOR XIO B3:0/0 XIO B3:0/2 BST XIC I:0.0/8 XIO B3:0/6 XIC B3:0/5 XIO B3:1/4 NXB XIO I:0.0/8 XIC I:0.0/10 BND XIO B3:2/0 XIO B3:2/1 XIO B3:1/15 XIO O:0.0/6 OTE O:0.0/5 EOR
%   B3:0/0  ENC_FLT %
%   B3:0/2  ENC_UP  "Cradle in highest position" %
%   I:0.0/8  AUTO  "Enter Auto Mode" %
%   B3:0/6  CRDL_LTCH2  "Send cradle down" %
%   B3:0/5  CRDL_LTCH1  "Send cradle up" %
%   B3:1/4  "Over Torque" %
%   I:0.0/10  CRDL_UP_SS  "Hand mode" %
%   B3:2/0  INFEED_CATCH  "Catch Infeed Barrier fault" %
%   B3:2/1  OUTFEED_CATCH  "Catch Outfeet Barrier Fault" %
%   B3:1/15  CRADLE_TIME_OUT  "Cradle movement Time Out" %
%   O:0.0/6  CRDL_DWN  "VFD REV" %
%   O:0.0/5  CRDL_UP  "VFD FWD" %
% Rung: 62 %
SOR XIO B3:0/0 XIO B3:0/1 BST XIC I:0.0/8 XIC B3:0/6 XIO B3:1/4 NXB XIO I:0.0/8 XIC I:0.0/9 BND XIO B3:2/0 XIO B3:2/1 XIO B3:2/3 XIO B3:1/10 XIO B3:1/15 XIO O:0.0/5 OTE O:0.0/6 EOR
%   B3:0/0  ENC_FLT %
%   B3:0/1  ENC_DOWN  "Cradle down position" %
%   I:0.0/8  AUTO  "Enter Auto Mode" %
%   B3:0/6  CRDL_LTCH2  "Send cradle down" %
%   B3:1/4  "Over Torque" %
%   I:0.0/9  CRDL_DWN_SS  "Hand mode" %
%   B3:2/0  INFEED_CATCH  "Catch Infeed Barrier fault" %
%   B3:2/1  OUTFEED_CATCH  "Catch Outfeet Barrier Fault" %
%   B3:2/3  DOWN_CATCH  "Cradle Down Overtravel" %
%   B3:1/10  "Lock cradle dowm" %
%   B3:1/15  CRADLE_TIME_OUT  "Cradle movement Time Out" %
%   O:0.0/5  CRDL_UP  "VFD FWD" %
%   O:0.0/6  CRDL_DWN  "VFD REV" %
% Rung: 63 %
SOR BST XIC O:0.0/5 NXB XIC O:0.0/6 BND OTE O:1.0/3 EOR
%   O:0.0/5  CRDL_UP  "VFD FWD" %
%   O:0.0/6  CRDL_DWN  "VFD REV" %
%   O:1.0/3  CRADLE_BREAK_CONTACT %
% Rung: 64 %
SOR XIC O:0.0/5 TON T4:15 1.0 5 0 EOR
%   O:0.0/5  CRDL_UP  "VFD FWD" %
%   T4:15  CRADLE_UP_TIMER %
% Rung: 65 %
SOR XIC O:0.0/6 TON T4:16 1.0 5 0 EOR
%   O:0.0/6  CRDL_DWN  "VFD REV" %
%   T4:16  CRADLE_DOWN_TIMER %

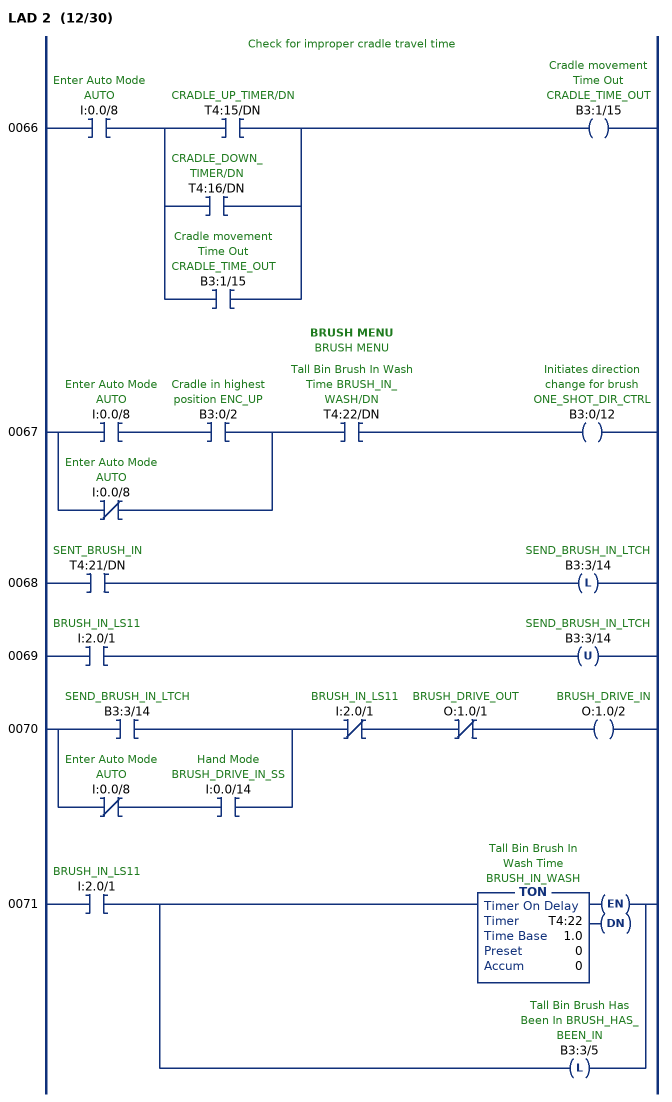
% Rung: 66 %
% Check for improper cradle travel time %
SOR XIC I:0.0/8 BST BST XIC T4:15/DN NXB XIC T4:16/DN BND NXB XIC B3:1/15 BND OTE B3:1/15 EOR
%   I:0.0/8  AUTO  "Enter Auto Mode" %
%   T4:15  CRADLE_UP_TIMER %
%   T4:16  CRADLE_DOWN_TIMER %
%   B3:1/15  CRADLE_TIME_OUT  "Cradle movement Time Out" %
% Rung: 67 %
% TITLE: BRUSH MENU %
% BRUSH MENU %
SOR BST XIC I:0.0/8 XIC B3:0/2 NXB XIO I:0.0/8 BND XIC T4:22/DN OTE B3:0/12 EOR
%   I:0.0/8  AUTO  "Enter Auto Mode" %
%   B3:0/2  ENC_UP  "Cradle in highest position" %
%   T4:22  BRUSH_IN_WASH  "Tall Bin Brush In Wash Time" %
%   B3:0/12  ONE_SHOT_DIR_CTRL  "Initiates direction change for brush" %
% Rung: 68 %
SOR XIC T4:21/DN OTL B3:3/14 EOR
%   T4:21/DN  SENT_BRUSH_IN %
%   B3:3/14  SEND_BRUSH_IN_LTCH %
% Rung: 69 %
SOR XIC I:2.0/1 OTU B3:3/14 EOR
%   I:2.0/1  BRUSH_IN_LS11 %
%   B3:3/14  SEND_BRUSH_IN_LTCH %
% Rung: 70 %
SOR BST XIC B3:3/14 NXB XIO I:0.0/8 XIC I:0.0/14 BND XIO I:2.0/1 XIO O:1.0/1 OTE O:1.0/2 EOR
%   B3:3/14  SEND_BRUSH_IN_LTCH %
%   I:0.0/8  AUTO  "Enter Auto Mode" %
%   I:0.0/14  BRUSH_DRIVE_IN_SS  "Hand Mode" %
%   I:2.0/1  BRUSH_IN_LS11 %
%   O:1.0/1  BRUSH_DRIVE_OUT %
%   O:1.0/2  BRUSH_DRIVE_IN %
% Rung: 71 %
SOR XIC I:2.0/1 BST TON T4:22 1.0 0 0 NXB OTL B3:3/5 BND EOR
%   I:2.0/1  BRUSH_IN_LS11 %
%   T4:22  BRUSH_IN_WASH  "Tall Bin Brush In Wash Time" %
%   B3:3/5  BRUSH_HAS_BEEN_IN  "Tall Bin Brush Has Been In" %

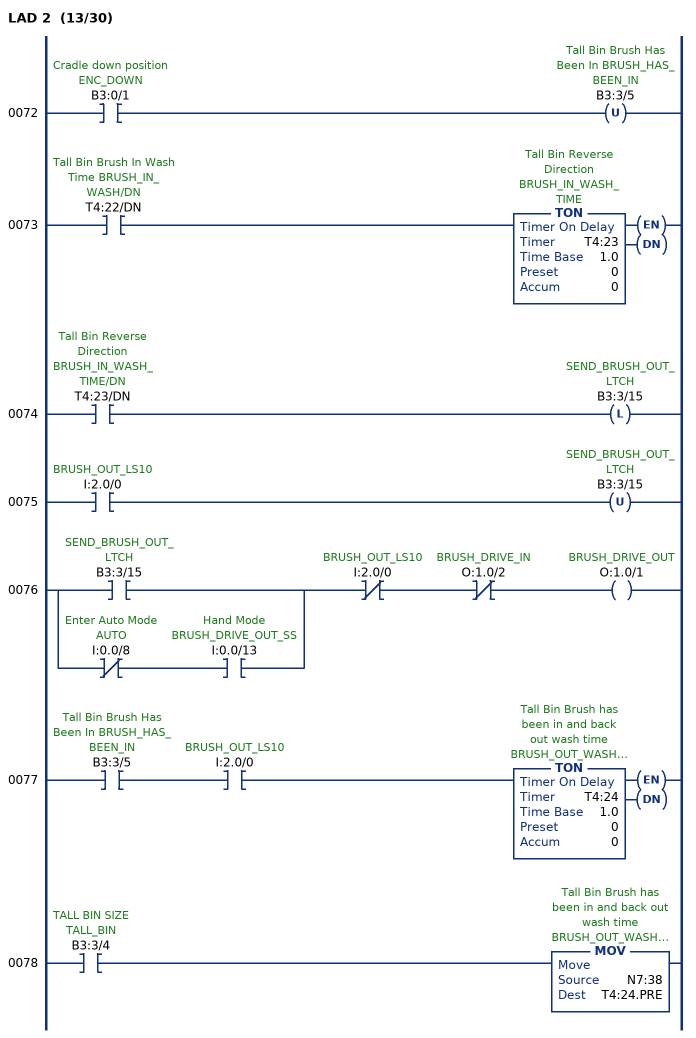
% Rung: 72 %
SOR XIC B3:0/1 OTU B3:3/5 EOR
%   B3:0/1  ENC_DOWN  "Cradle down position" %
%   B3:3/5  BRUSH_HAS_BEEN_IN  "Tall Bin Brush Has Been In" %
% Rung: 73 %
SOR XIC T4:22/DN TON T4:23 1.0 0 0 EOR
%   T4:22  BRUSH_IN_WASH  "Tall Bin Brush In Wash Time" %
%   T4:23  BRUSH_IN_WASH_TIME  "Tall Bin Reverse Direction" %
% Rung: 74 %
SOR XIC T4:23/DN OTL B3:3/15 EOR
%   T4:23  BRUSH_IN_WASH_TIME  "Tall Bin Reverse Direction" %
%   B3:3/15  SEND_BRUSH_OUT_LTCH %
% Rung: 75 %
SOR XIC I:2.0/0 OTU B3:3/15 EOR
%   I:2.0/0  BRUSH_OUT_LS10 %
%   B3:3/15  SEND_BRUSH_OUT_LTCH %
% Rung: 76 %
SOR BST XIC B3:3/15 NXB XIO I:0.0/8 XIC I:0.0/13 BND XIO I:2.0/0 XIO O:1.0/2 OTE O:1.0/1 EOR
%   B3:3/15  SEND_BRUSH_OUT_LTCH %
%   I:0.0/8  AUTO  "Enter Auto Mode" %
%   I:0.0/13  BRUSH_DRIVE_OUT_SS  "Hand Mode" %
%   I:2.0/0  BRUSH_OUT_LS10 %
%   O:1.0/2  BRUSH_DRIVE_IN %
%   O:1.0/1  BRUSH_DRIVE_OUT %
% Rung: 77 %
SOR XIC B3:3/5 XIC I:2.0/0 TON T4:24 1.0 0 0 EOR
%   B3:3/5  BRUSH_HAS_BEEN_IN  "Tall Bin Brush Has Been In" %
%   I:2.0/0  BRUSH_OUT_LS10 %
%   T4:24  BRUSH_OUT_WASH_TIME  "Tall Bin Brush has been in and back out wash time" %
% Rung: 78 %
SOR XIC B3:3/4 MOV N7:38 T4:24.PRE EOR
%   B3:3/4  TALL_BIN  "TALL BIN SIZE" %
%   N7:38  TALLBIN_BRUSH_TIME  "HMI Tall Bin Brush Time" %
%   T4:24  BRUSH_OUT_WASH_TIME  "Tall Bin Brush has been in and back out wash time" %

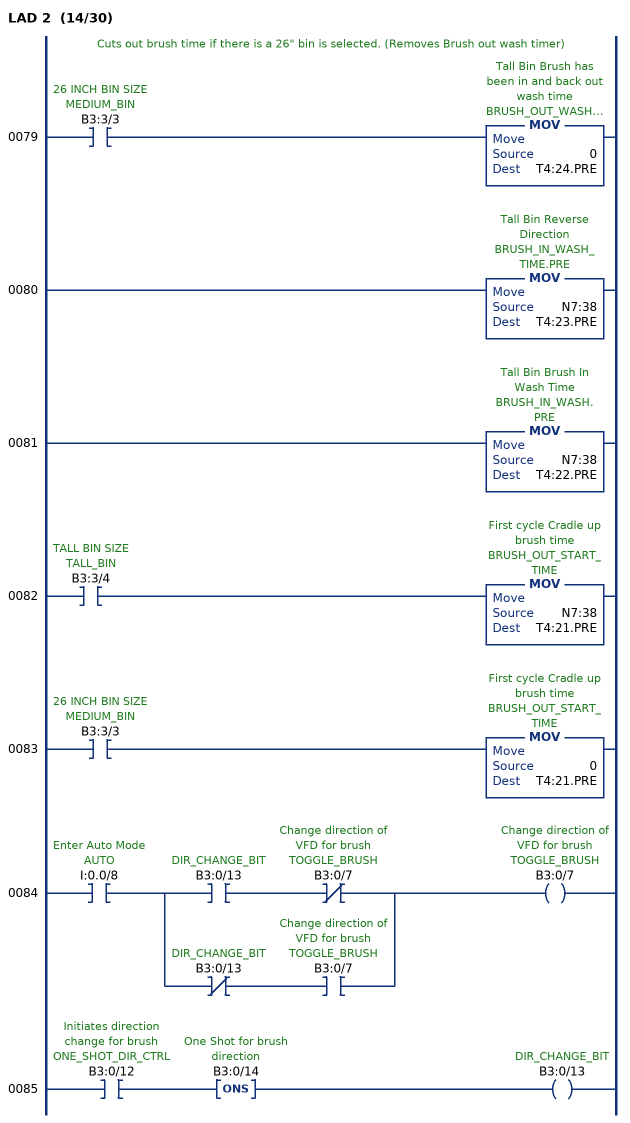
% Rung: 79 %
% Cuts out brush time if there is a 26" bin is selected. (Removes Brush out wash timer) %
SOR XIC B3:3/3 MOV 0 T4:24.PRE EOR
%   B3:3/3  MEDIUM_BIN  "26 INCH BIN SIZE" %
%   T4:24  BRUSH_OUT_WASH_TIME  "Tall Bin Brush has been in and back out wash time" %
% Rung: 80 %
SOR MOV N7:38 T4:23.PRE EOR
%   N7:38  TALLBIN_BRUSH_TIME  "HMI Tall Bin Brush Time" %
%   T4:23  BRUSH_IN_WASH_TIME  "Tall Bin Reverse Direction" %
% Rung: 81 %
SOR MOV N7:38 T4:22.PRE EOR
%   N7:38  TALLBIN_BRUSH_TIME  "HMI Tall Bin Brush Time" %
%   T4:22  BRUSH_IN_WASH  "Tall Bin Brush In Wash Time" %
% Rung: 82 %
SOR XIC B3:3/4 MOV N7:38 T4:21.PRE EOR
%   B3:3/4  TALL_BIN  "TALL BIN SIZE" %
%   N7:38  TALLBIN_BRUSH_TIME  "HMI Tall Bin Brush Time" %
%   T4:21.PRE  BRUSH_OUT_START_TIME  "First cycle Cradle up brush time" %
% Rung: 83 %
SOR XIC B3:3/3 MOV 0 T4:21.PRE EOR
%   B3:3/3  MEDIUM_BIN  "26 INCH BIN SIZE" %
%   T4:21.PRE  BRUSH_OUT_START_TIME  "First cycle Cradle up brush time" %
% Rung: 84 %
SOR XIC I:0.0/8 BST XIC B3:0/13 XIO B3:0/7 NXB XIO B3:0/13 XIC B3:0/7 BND OTE B3:0/7 EOR
%   I:0.0/8  AUTO  "Enter Auto Mode" %
%   B3:0/13  DIR_CHANGE_BIT %
%   B3:0/7  TOGGLE_BRUSH  "Change direction of VFD for brush" %
% Rung: 85 %
SOR XIC B3:0/12 ONS B3:0/14 OTE B3:0/13 EOR
%   B3:0/12  ONE_SHOT_DIR_CTRL  "Initiates direction change for brush" %
%   B3:0/14  "One Shot for brush direction" %
%   B3:0/13  DIR_CHANGE_BIT %

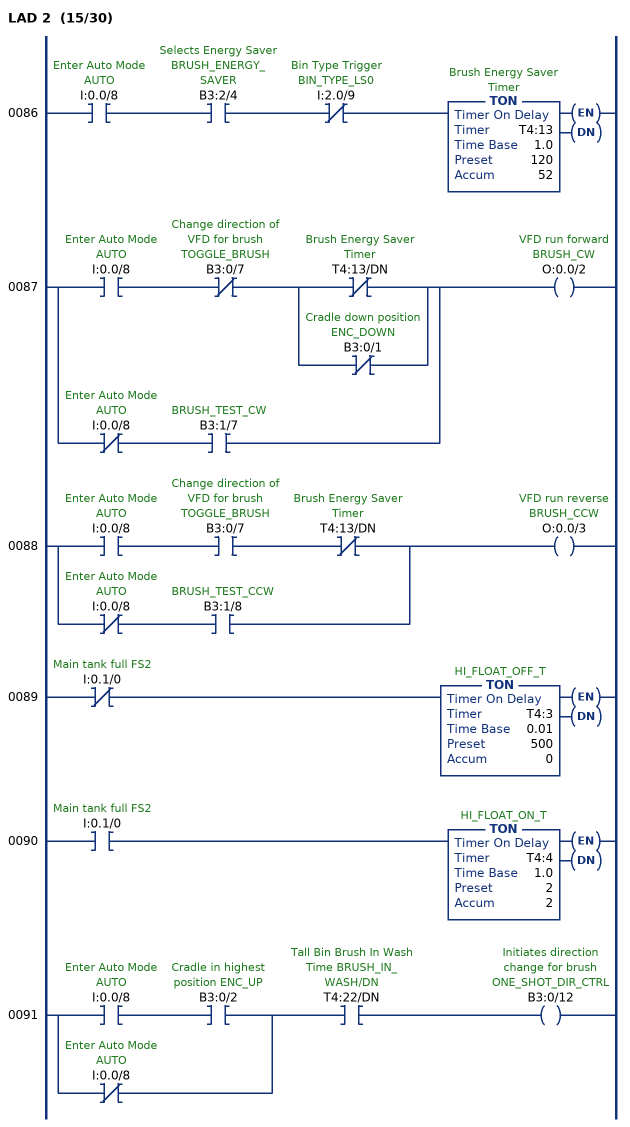
% Rung: 86 %
SOR XIC I:0.0/8 XIC B3:2/4 XIO I:2.0/9 TON T4:13 1.0 120 52 EOR
%   I:0.0/8  AUTO  "Enter Auto Mode" %
%   B3:2/4  BRUSH_ENERGY_SAVER  "Selects Energy Saver" %
%   I:2.0/9  BIN_TYPE_LS0  "Bin Type Trigger" %
%   T4:13  "Brush Energy Saver Timer" %
% Rung: 87 %
SOR BST XIC I:0.0/8 XIO B3:0/7 BST XIO T4:13/DN NXB XIO B3:0/1 BND NXB XIO I:0.0/8 XIC B3:1/7 BND OTE O:0.0/2 EOR
%   I:0.0/8  AUTO  "Enter Auto Mode" %
%   B3:0/7  TOGGLE_BRUSH  "Change direction of VFD for brush" %
%   T4:13  "Brush Energy Saver Timer" %
%   B3:0/1  ENC_DOWN  "Cradle down position" %
%   B3:1/7  BRUSH_TEST_CW %
%   O:0.0/2  BRUSH_CW  "VFD run forward" %
% Rung: 88 %
SOR BST XIC I:0.0/8 XIC B3:0/7 XIO T4:13/DN NXB XIO I:0.0/8 XIC B3:1/8 BND OTE O:0.0/3 EOR
%   I:0.0/8  AUTO  "Enter Auto Mode" %
%   B3:0/7  TOGGLE_BRUSH  "Change direction of VFD for brush" %
%   T4:13  "Brush Energy Saver Timer" %
%   B3:1/8  BRUSH_TEST_CCW %
%   O:0.0/3  BRUSH_CCW  "VFD run reverse" %
% Rung: 89 %
SOR XIO I:0.1/0 TON T4:3 0.01 500 0 EOR
%   I:0.1/0  FS2  "Main tank full" %
%   T4:3  HI_FLOAT_OFF_T %
% Rung: 90 %
SOR XIC I:0.1/0 TON T4:4 1.0 2 2 EOR
%   I:0.1/0  FS2  "Main tank full" %
%   T4:4  HI_FLOAT_ON_T %
% Rung: 91 %
SOR BST XIC I:0.0/8 XIC B3:0/2 NXB XIO I:0.0/8 BND XIC T4:22/DN OTE B3:0/12 EOR
%   I:0.0/8  AUTO  "Enter Auto Mode" %
%   B3:0/2  ENC_UP  "Cradle in highest position" %
%   T4:22  BRUSH_IN_WASH  "Tall Bin Brush In Wash Time" %
%   B3:0/12  ONE_SHOT_DIR_CTRL  "Initiates direction change for brush" %

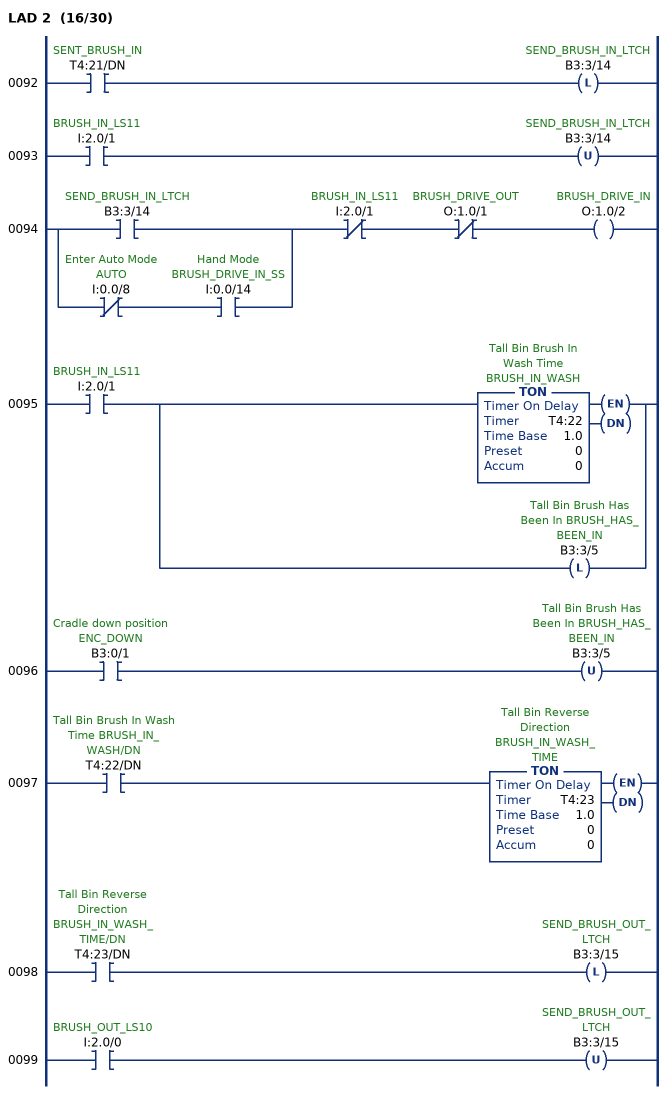
% Rung: 92 %
SOR XIC T4:21/DN OTL B3:3/14 EOR
%   T4:21/DN  SENT_BRUSH_IN %
%   B3:3/14  SEND_BRUSH_IN_LTCH %
% Rung: 93 %
SOR XIC I:2.0/1 OTU B3:3/14 EOR
%   I:2.0/1  BRUSH_IN_LS11 %
%   B3:3/14  SEND_BRUSH_IN_LTCH %
% Rung: 94 %
SOR BST XIC B3:3/14 NXB XIO I:0.0/8 XIC I:0.0/14 BND XIO I:2.0/1 XIO O:1.0/1 OTE O:1.0/2 EOR
%   B3:3/14  SEND_BRUSH_IN_LTCH %
%   I:0.0/8  AUTO  "Enter Auto Mode" %
%   I:0.0/14  BRUSH_DRIVE_IN_SS  "Hand Mode" %
%   I:2.0/1  BRUSH_IN_LS11 %
%   O:1.0/1  BRUSH_DRIVE_OUT %
%   O:1.0/2  BRUSH_DRIVE_IN %
% Rung: 95 %
SOR XIC I:2.0/1 BST TON T4:22 1.0 0 0 NXB OTL B3:3/5 BND EOR
%   I:2.0/1  BRUSH_IN_LS11 %
%   T4:22  BRUSH_IN_WASH  "Tall Bin Brush In Wash Time" %
%   B3:3/5  BRUSH_HAS_BEEN_IN  "Tall Bin Brush Has Been In" %
% Rung: 96 %
SOR XIC B3:0/1 OTU B3:3/5 EOR
%   B3:0/1  ENC_DOWN  "Cradle down position" %
%   B3:3/5  BRUSH_HAS_BEEN_IN  "Tall Bin Brush Has Been In" %
% Rung: 97 %
SOR XIC T4:22/DN TON T4:23 1.0 0 0 EOR
%   T4:22  BRUSH_IN_WASH  "Tall Bin Brush In Wash Time" %
%   T4:23  BRUSH_IN_WASH_TIME  "Tall Bin Reverse Direction" %
% Rung: 98 %
SOR XIC T4:23/DN OTL B3:3/15 EOR
%   T4:23  BRUSH_IN_WASH_TIME  "Tall Bin Reverse Direction" %
%   B3:3/15  SEND_BRUSH_OUT_LTCH %
% Rung: 99 %
SOR XIC I:2.0/0 OTU B3:3/15 EOR
%   I:2.0/0  BRUSH_OUT_LS10 %
%   B3:3/15  SEND_BRUSH_OUT_LTCH %

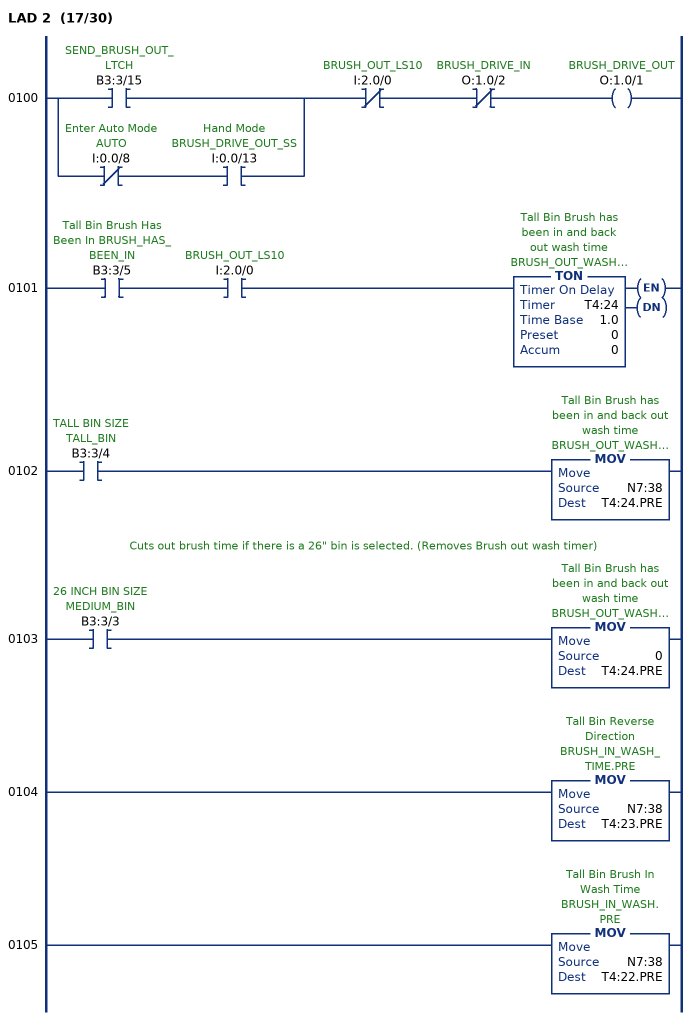
% Rung: 100 %
SOR BST XIC B3:3/15 NXB XIO I:0.0/8 XIC I:0.0/13 BND XIO I:2.0/0 XIO O:1.0/2 OTE O:1.0/1 EOR
%   B3:3/15  SEND_BRUSH_OUT_LTCH %
%   I:0.0/8  AUTO  "Enter Auto Mode" %
%   I:0.0/13  BRUSH_DRIVE_OUT_SS  "Hand Mode" %
%   I:2.0/0  BRUSH_OUT_LS10 %
%   O:1.0/2  BRUSH_DRIVE_IN %
%   O:1.0/1  BRUSH_DRIVE_OUT %
% Rung: 101 %
SOR XIC B3:3/5 XIC I:2.0/0 TON T4:24 1.0 0 0 EOR
%   B3:3/5  BRUSH_HAS_BEEN_IN  "Tall Bin Brush Has Been In" %
%   I:2.0/0  BRUSH_OUT_LS10 %
%   T4:24  BRUSH_OUT_WASH_TIME  "Tall Bin Brush has been in and back out wash time" %
% Rung: 102 %
SOR XIC B3:3/4 MOV N7:38 T4:24.PRE EOR
%   B3:3/4  TALL_BIN  "TALL BIN SIZE" %
%   N7:38  TALLBIN_BRUSH_TIME  "HMI Tall Bin Brush Time" %
%   T4:24  BRUSH_OUT_WASH_TIME  "Tall Bin Brush has been in and back out wash time" %
% Rung: 103 %
% Cuts out brush time if there is a 26" bin is selected. (Removes Brush out wash timer) %
SOR XIC B3:3/3 MOV 0 T4:24.PRE EOR
%   B3:3/3  MEDIUM_BIN  "26 INCH BIN SIZE" %
%   T4:24  BRUSH_OUT_WASH_TIME  "Tall Bin Brush has been in and back out wash time" %
% Rung: 104 %
SOR MOV N7:38 T4:23.PRE EOR
%   N7:38  TALLBIN_BRUSH_TIME  "HMI Tall Bin Brush Time" %
%   T4:23  BRUSH_IN_WASH_TIME  "Tall Bin Reverse Direction" %
% Rung: 105 %
SOR MOV N7:38 T4:22.PRE EOR
%   N7:38  TALLBIN_BRUSH_TIME  "HMI Tall Bin Brush Time" %
%   T4:22  BRUSH_IN_WASH  "Tall Bin Brush In Wash Time" %

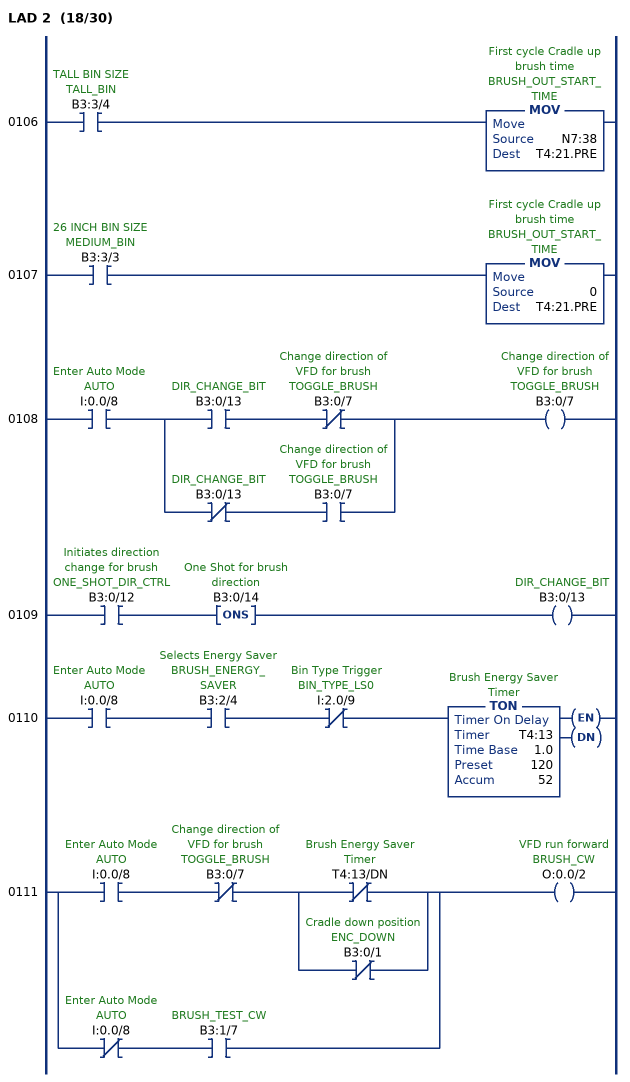
% Rung: 106 %
SOR XIC B3:3/4 MOV N7:38 T4:21.PRE EOR
%   B3:3/4  TALL_BIN  "TALL BIN SIZE" %
%   N7:38  TALLBIN_BRUSH_TIME  "HMI Tall Bin Brush Time" %
%   T4:21.PRE  BRUSH_OUT_START_TIME  "First cycle Cradle up brush time" %
% Rung: 107 %
SOR XIC B3:3/3 MOV 0 T4:21.PRE EOR
%   B3:3/3  MEDIUM_BIN  "26 INCH BIN SIZE" %
%   T4:21.PRE  BRUSH_OUT_START_TIME  "First cycle Cradle up brush time" %
% Rung: 108 %
SOR XIC I:0.0/8 BST XIC B3:0/13 XIO B3:0/7 NXB XIO B3:0/13 XIC B3:0/7 BND OTE B3:0/7 EOR
%   I:0.0/8  AUTO  "Enter Auto Mode" %
%   B3:0/13  DIR_CHANGE_BIT %
%   B3:0/7  TOGGLE_BRUSH  "Change direction of VFD for brush" %
% Rung: 109 %
SOR XIC B3:0/12 ONS B3:0/14 OTE B3:0/13 EOR
%   B3:0/12  ONE_SHOT_DIR_CTRL  "Initiates direction change for brush" %
%   B3:0/14  "One Shot for brush direction" %
%   B3:0/13  DIR_CHANGE_BIT %
% Rung: 110 %
SOR XIC I:0.0/8 XIC B3:2/4 XIO I:2.0/9 TON T4:13 1.0 120 52 EOR
%   I:0.0/8  AUTO  "Enter Auto Mode" %
%   B3:2/4  BRUSH_ENERGY_SAVER  "Selects Energy Saver" %
%   I:2.0/9  BIN_TYPE_LS0  "Bin Type Trigger" %
%   T4:13  "Brush Energy Saver Timer" %
% Rung: 111 %
SOR BST XIC I:0.0/8 XIO B3:0/7 BST XIO T4:13/DN NXB XIO B3:0/1 BND NXB XIO I:0.0/8 XIC B3:1/7 BND OTE O:0.0/2 EOR
%   I:0.0/8  AUTO  "Enter Auto Mode" %
%   B3:0/7  TOGGLE_BRUSH  "Change direction of VFD for brush" %
%   T4:13  "Brush Energy Saver Timer" %
%   B3:0/1  ENC_DOWN  "Cradle down position" %
%   B3:1/7  BRUSH_TEST_CW %
%   O:0.0/2  BRUSH_CW  "VFD run forward" %

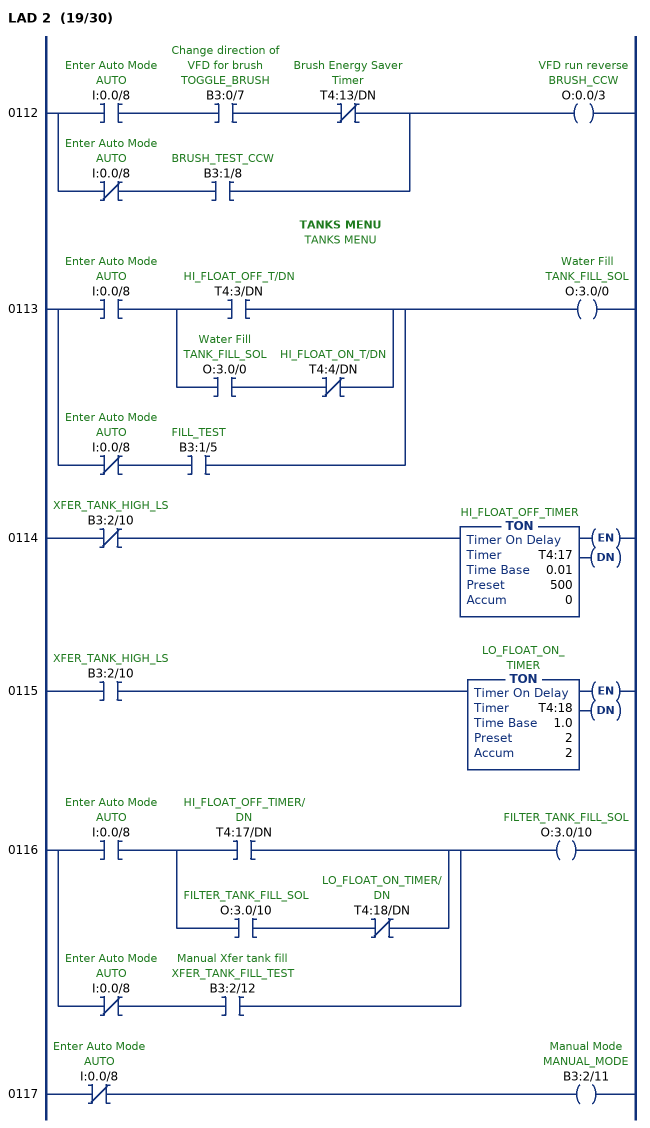
% Rung: 112 %
SOR BST XIC I:0.0/8 XIC B3:0/7 XIO T4:13/DN NXB XIO I:0.0/8 XIC B3:1/8 BND OTE O:0.0/3 EOR
%   I:0.0/8  AUTO  "Enter Auto Mode" %
%   B3:0/7  TOGGLE_BRUSH  "Change direction of VFD for brush" %
%   T4:13  "Brush Energy Saver Timer" %
%   B3:1/8  BRUSH_TEST_CCW %
%   O:0.0/3  BRUSH_CCW  "VFD run reverse" %
% Rung: 113 %
% TITLE: TANKS MENU %
% TANKS MENU %
SOR BST XIC I:0.0/8 BST XIC T4:3/DN NXB XIC O:3.0/0 XIO T4:4/DN BND NXB XIO I:0.0/8 XIC B3:1/5 BND OTE O:3.0/0 EOR
%   I:0.0/8  AUTO  "Enter Auto Mode" %
%   T4:3  HI_FLOAT_OFF_T %
%   O:3.0/0  TANK_FILL_SOL  "Water Fill" %
%   T4:4  HI_FLOAT_ON_T %
%   B3:1/5  FILL_TEST %
% Rung: 114 %
SOR XIO B3:2/10 TON T4:17 0.01 500 0 EOR
%   B3:2/10  XFER_TANK_HIGH_LS %
%   T4:17  HI_FLOAT_OFF_TIMER %
% Rung: 115 %
SOR XIC B3:2/10 TON T4:18 1.0 2 2 EOR
%   B3:2/10  XFER_TANK_HIGH_LS %
%   T4:18  LO_FLOAT_ON_TIMER %
% Rung: 116 %
SOR BST XIC I:0.0/8 BST XIC T4:17/DN NXB XIC O:3.0/10 XIO T4:18/DN BND NXB XIO I:0.0/8 XIC B3:2/12 BND OTE O:3.0/10 EOR
%   I:0.0/8  AUTO  "Enter Auto Mode" %
%   T4:17  HI_FLOAT_OFF_TIMER %
%   O:3.0/10  FILTER_TANK_FILL_SOL %
%   T4:18  LO_FLOAT_ON_TIMER %
%   B3:2/12  XFER_TANK_FILL_TEST  "Manual Xfer tank fill" %
% Rung: 117 %
SOR XIO I:0.0/8 OTE B3:2/11 EOR
%   I:0.0/8  AUTO  "Enter Auto Mode" %
%   B3:2/11  MANUAL_MODE  "Manual Mode" %

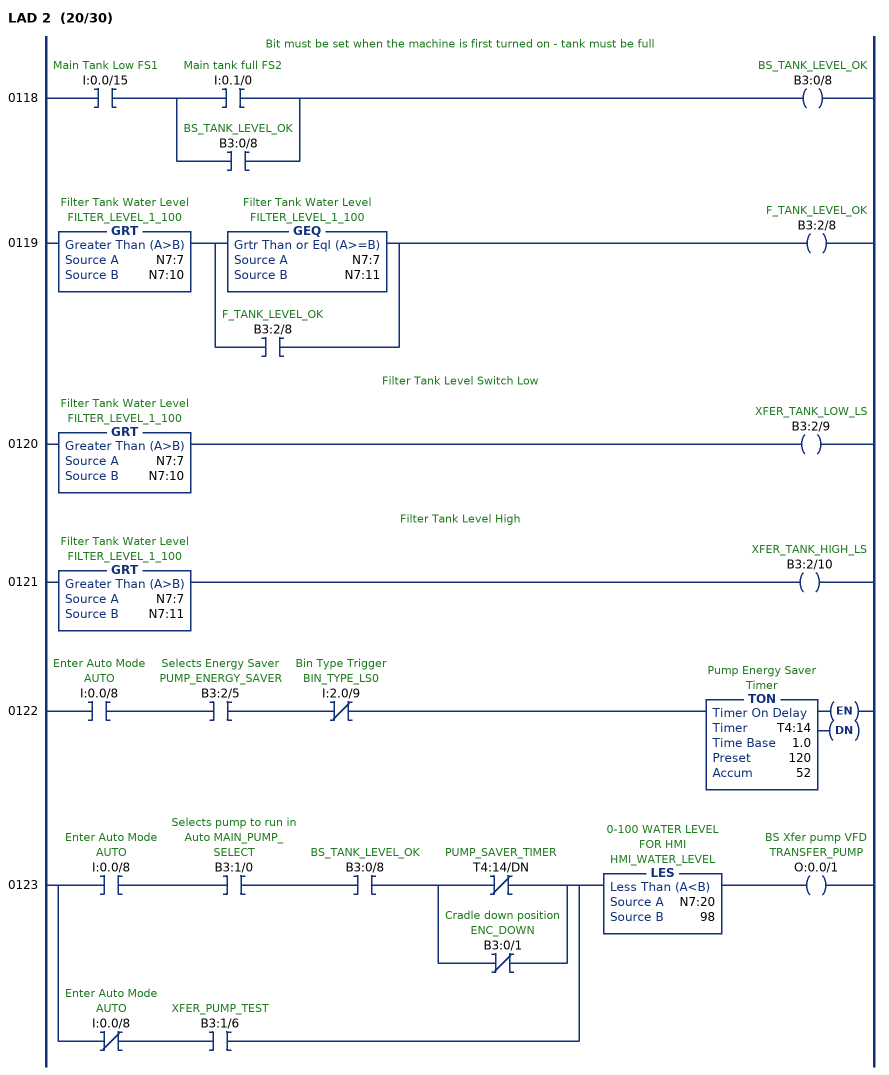
% Rung: 118 %
% Bit must be set when the machine is first turned on - tank must be full %
SOR XIC I:0.0/15 BST XIC I:0.1/0 NXB XIC B3:0/8 BND OTE B3:0/8 EOR
%   I:0.0/15  FS1  "Main Tank Low" %
%   I:0.1/0  FS2  "Main tank full" %
%   B3:0/8  BS_TANK_LEVEL_OK %
% Rung: 119 %
SOR GRT N7:7 N7:10 BST GEQ N7:7 N7:11 NXB XIC B3:2/8 BND OTE B3:2/8 EOR
%   N7:7  FILTER_LEVEL_1_100  "Filter Tank Water Level" %
%   N7:10  FILTER_LOW_LS  "Filter Tank Low Level LS" %
%   N7:11  FILTER_TANK_FULL_LS  "Filter Tank High Water LS" %
%   B3:2/8  F_TANK_LEVEL_OK %
% Rung: 120 %
% Filter Tank Level Switch Low %
SOR GRT N7:7 N7:10 OTE B3:2/9 EOR
%   N7:7  FILTER_LEVEL_1_100  "Filter Tank Water Level" %
%   N7:10  FILTER_LOW_LS  "Filter Tank Low Level LS" %
%   B3:2/9  XFER_TANK_LOW_LS %
% Rung: 121 %
% Filter Tank Level High %
SOR GRT N7:7 N7:11 OTE B3:2/10 EOR
%   N7:7  FILTER_LEVEL_1_100  "Filter Tank Water Level" %
%   N7:11  FILTER_TANK_FULL_LS  "Filter Tank High Water LS" %
%   B3:2/10  XFER_TANK_HIGH_LS %
% Rung: 122 %
SOR XIC I:0.0/8 XIC B3:2/5 XIO I:2.0/9 TON T4:14 1.0 120 52 EOR
%   I:0.0/8  AUTO  "Enter Auto Mode" %
%   B3:2/5  PUMP_ENERGY_SAVER  "Selects Energy Saver" %
%   I:2.0/9  BIN_TYPE_LS0  "Bin Type Trigger" %
%   T4:14  "Pump Energy Saver Timer" %
% Rung: 123 %
SOR BST XIC I:0.0/8 XIC B3:1/0 XIC B3:0/8 BST XIO T4:14/DN NXB XIO B3:0/1 BND NXB XIO I:0.0/8 XIC B3:1/6 BND LES N7:20 98 OTE O:0.0/1 EOR
%   I:0.0/8  AUTO  "Enter Auto Mode" %
%   B3:1/0  MAIN_PUMP_SELECT  "Selects pump to run in Auto" %
%   B3:0/8  BS_TANK_LEVEL_OK %
%   T4:14/DN  PUMP_SAVER_TIMER %
%   B3:0/1  ENC_DOWN  "Cradle down position" %
%   B3:1/6  XFER_PUMP_TEST %
%   N7:20  HMI_WATER_LEVEL  "0-100 WATER LEVEL FOR HMI" %
%   O:0.0/1  TRANSFER_PUMP  "BS Xfer pump VFD" %

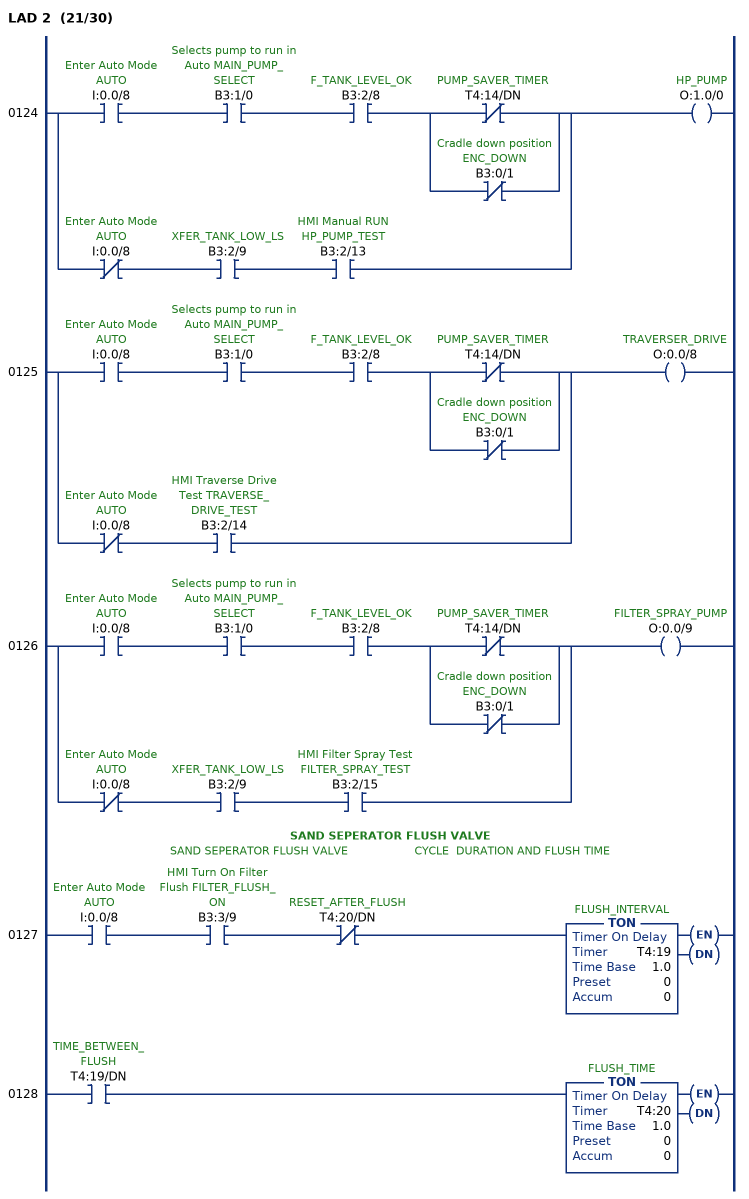
% Rung: 124 %
SOR BST XIC I:0.0/8 XIC B3:1/0 XIC B3:2/8 BST XIO T4:14/DN NXB XIO B3:0/1 BND NXB XIO I:0.0/8 XIC B3:2/9 XIC B3:2/13 BND OTE O:1.0/0 EOR
%   I:0.0/8  AUTO  "Enter Auto Mode" %
%   B3:1/0  MAIN_PUMP_SELECT  "Selects pump to run in Auto" %
%   B3:2/8  F_TANK_LEVEL_OK %
%   T4:14/DN  PUMP_SAVER_TIMER %
%   B3:0/1  ENC_DOWN  "Cradle down position" %
%   B3:2/9  XFER_TANK_LOW_LS %
%   B3:2/13  HP_PUMP_TEST  "HMI Manual RUN" %
%   O:1.0/0  HP_PUMP %
% Rung: 125 %
SOR BST XIC I:0.0/8 XIC B3:1/0 XIC B3:2/8 BST XIO T4:14/DN NXB XIO B3:0/1 BND NXB XIO I:0.0/8 XIC B3:2/14 BND OTE O:0.0/8 EOR
%   I:0.0/8  AUTO  "Enter Auto Mode" %
%   B3:1/0  MAIN_PUMP_SELECT  "Selects pump to run in Auto" %
%   B3:2/8  F_TANK_LEVEL_OK %
%   T4:14/DN  PUMP_SAVER_TIMER %
%   B3:0/1  ENC_DOWN  "Cradle down position" %
%   B3:2/14  TRAVERSE_DRIVE_TEST  "HMI Traverse Drive Test" %
%   O:0.0/8  TRAVERSER_DRIVE %
% Rung: 126 %
SOR BST XIC I:0.0/8 XIC B3:1/0 XIC B3:2/8 BST XIO T4:14/DN NXB XIO B3:0/1 BND NXB XIO I:0.0/8 XIC B3:2/9 XIC B3:2/15 BND OTE O:0.0/9 EOR
%   I:0.0/8  AUTO  "Enter Auto Mode" %
%   B3:1/0  MAIN_PUMP_SELECT  "Selects pump to run in Auto" %
%   B3:2/8  F_TANK_LEVEL_OK %
%   T4:14/DN  PUMP_SAVER_TIMER %
%   B3:0/1  ENC_DOWN  "Cradle down position" %
%   B3:2/9  XFER_TANK_LOW_LS %
%   B3:2/15  FILTER_SPRAY_TEST  "HMI Filter Spray Test" %
%   O:0.0/9  FILTER_SPRAY_PUMP %
% Rung: 127 %
% TITLE: SAND SEPERATOR FLUSH VALVE %
% SAND SEPERATOR FLUSH VALVE                   CYCLE  DURATION AND FLUSH TIME %
SOR XIC I:0.0/8 XIC B3:3/9 XIO T4:20/DN TON T4:19 1.0 0 0 EOR
%   I:0.0/8  AUTO  "Enter Auto Mode" %
%   B3:3/9  FILTER_FLUSH_ON  "HMI Turn On Filter Flush" %
%   T4:20/DN  RESET_AFTER_FLUSH %
%   T4:19  FLUSH_INTERVAL %
% Rung: 128 %
SOR XIC T4:19/DN TON T4:20 1.0 0 0 EOR
%   T4:19/DN  TIME_BETWEEN_FLUSH %
%   T4:20  FLUSH_TIME %

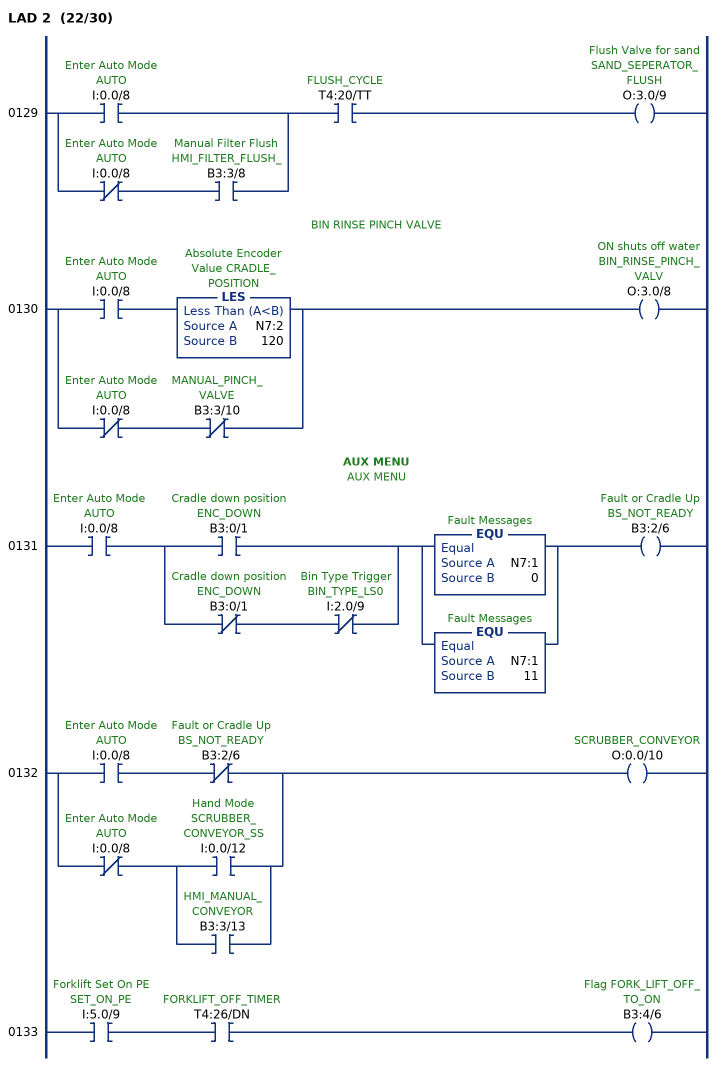
% Rung: 129 %
SOR BST XIC I:0.0/8 NXB XIO I:0.0/8 XIC B3:3/8 BND XIC T4:20/TT OTE O:3.0/9 EOR
%   I:0.0/8  AUTO  "Enter Auto Mode" %
%   B3:3/8  HMI_FILTER_FLUSH_  "Manual Filter Flush" %
%   T4:20/TT  FLUSH_CYCLE %
%   O:3.0/9  SAND_SEPERATOR_FLUSH  "Flush Valve for sand" %
% Rung: 130 %
% BIN RINSE PINCH VALVE %
SOR BST XIC I:0.0/8 LES N7:2 120 NXB XIO I:0.0/8 XIO B3:3/10 BND OTE O:3.0/8 EOR
%   I:0.0/8  AUTO  "Enter Auto Mode" %
%   N7:2  CRADLE_POSITION  "Absolute Encoder Value" %
%   B3:3/10  MANUAL_PINCH_VALVE %
%   O:3.0/8  BIN_RINSE_PINCH_VALV  "ON shuts off water" %
% Rung: 131 %
% TITLE: AUX MENU %
% AUX MENU %
SOR XIC I:0.0/8 BST XIC B3:0/1 NXB XIO B3:0/1 XIO I:2.0/9 BND BST EQU N7:1 0 NXB EQU N7:1 11 BND OTE B3:2/6 EOR
%   I:0.0/8  AUTO  "Enter Auto Mode" %
%   B3:0/1  ENC_DOWN  "Cradle down position" %
%   I:2.0/9  BIN_TYPE_LS0  "Bin Type Trigger" %
%   N7:1  "Fault Messages" %
%   B3:2/6  BS_NOT_READY  "Fault or Cradle Up" %
% Rung: 132 %
SOR BST XIC I:0.0/8 XIO B3:2/6 NXB XIO I:0.0/8 BST XIC I:0.0/12 NXB XIC B3:3/13 BND BND OTE O:0.0/10 EOR
%   I:0.0/8  AUTO  "Enter Auto Mode" %
%   B3:2/6  BS_NOT_READY  "Fault or Cradle Up" %
%   I:0.0/12  SCRUBBER_CONVEYOR_SS  "Hand Mode" %
%   B3:3/13  HMI_MANUAL_CONVEYOR %
%   O:0.0/10  SCRUBBER_CONVEYOR %
% Rung: 133 %
SOR XIC I:5.0/9 XIC T4:26/DN OTE B3:4/6 EOR
%   I:5.0/9  SET_ON_PE  "Forklift Set On PE" %
%   T4:26/DN  FORKLIFT_OFF_TIMER %
%   B3:4/6  FORK_LIFT_OFF_TO_ON  "Flag" %

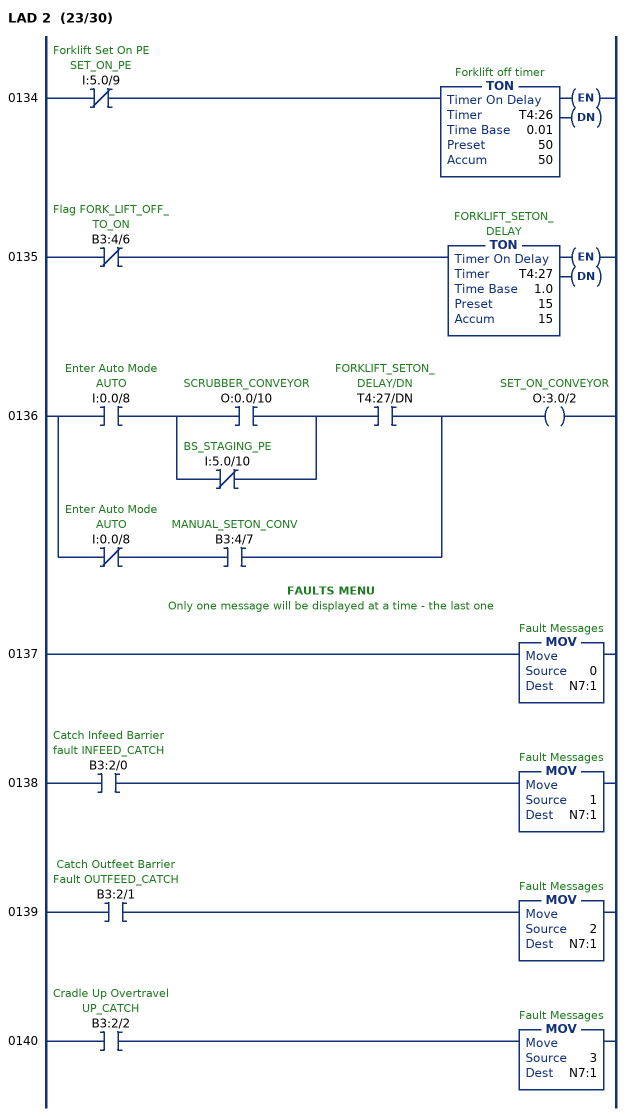
% Rung: 134 %
SOR XIO I:5.0/9 TON T4:26 0.01 50 50 EOR
%   I:5.0/9  SET_ON_PE  "Forklift Set On PE" %
%   T4:26  "Forklift off timer" %
% Rung: 135 %
SOR XIO B3:4/6 TON T4:27 1.0 15 15 EOR
%   B3:4/6  FORK_LIFT_OFF_TO_ON  "Flag" %
%   T4:27  FORKLIFT_SETON_DELAY %
% Rung: 136 %
SOR BST XIC I:0.0/8 BST XIC O:0.0/10 NXB XIO I:5.0/10 BND XIC T4:27/DN NXB XIO I:0.0/8 XIC B3:4/7 BND OTE O:3.0/2 EOR
%   I:0.0/8  AUTO  "Enter Auto Mode" %
%   O:0.0/10  SCRUBBER_CONVEYOR %
%   I:5.0/10  BS_STAGING_PE %
%   T4:27  FORKLIFT_SETON_DELAY %
%   B3:4/7  MANUAL_SETON_CONV %
%   O:3.0/2  SET_ON_CONVEYOR %
% Rung: 137 %
% TITLE: FAULTS MENU %
% Only one message will be displayed at a time - the last one %
SOR MOV 0 N7:1 EOR
%   N7:1  "Fault Messages" %
% Rung: 138 %
SOR XIC B3:2/0 MOV 1 N7:1 EOR
%   B3:2/0  INFEED_CATCH  "Catch Infeed Barrier fault" %
%   N7:1  "Fault Messages" %
% Rung: 139 %
SOR XIC B3:2/1 MOV 2 N7:1 EOR
%   B3:2/1  OUTFEED_CATCH  "Catch Outfeet Barrier Fault" %
%   N7:1  "Fault Messages" %
% Rung: 140 %
SOR XIC B3:2/2 MOV 3 N7:1 EOR
%   B3:2/2  UP_CATCH  "Cradle Up Overtravel" %
%   N7:1  "Fault Messages" %

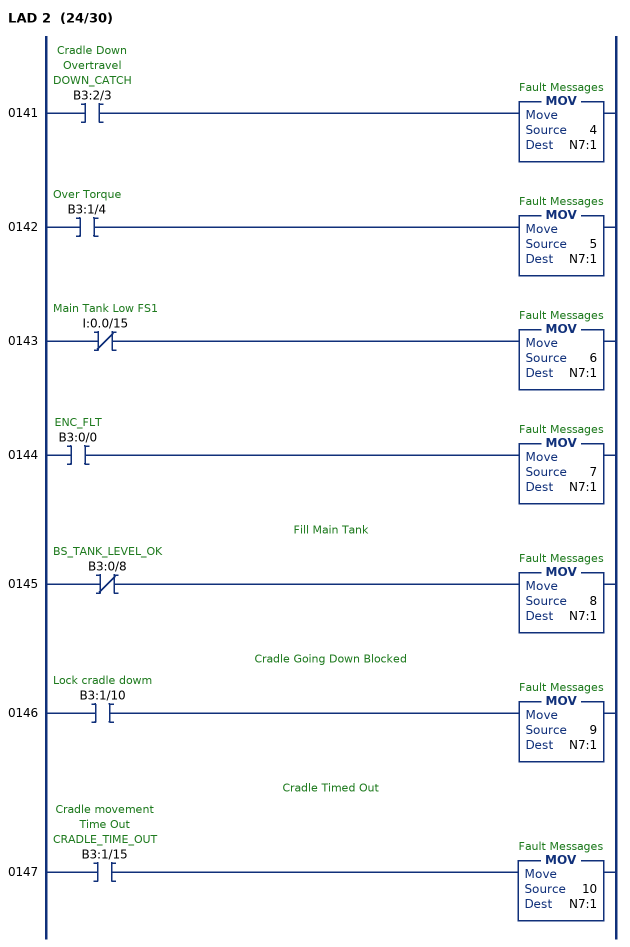
% Rung: 141 %
SOR XIC B3:2/3 MOV 4 N7:1 EOR
%   B3:2/3  DOWN_CATCH  "Cradle Down Overtravel" %
%   N7:1  "Fault Messages" %
% Rung: 142 %
SOR XIC B3:1/4 MOV 5 N7:1 EOR
%   B3:1/4  "Over Torque" %
%   N7:1  "Fault Messages" %
% Rung: 143 %
SOR XIO I:0.0/15 MOV 6 N7:1 EOR
%   I:0.0/15  FS1  "Main Tank Low" %
%   N7:1  "Fault Messages" %
% Rung: 144 %
SOR XIC B3:0/0 MOV 7 N7:1 EOR
%   B3:0/0  ENC_FLT %
%   N7:1  "Fault Messages" %
% Rung: 145 %
% Fill Main Tank %
SOR XIO B3:0/8 MOV 8 N7:1 EOR
%   B3:0/8  BS_TANK_LEVEL_OK %
%   N7:1  "Fault Messages" %
% Rung: 146 %
% Cradle Going Down Blocked %
SOR XIC B3:1/10 MOV 9 N7:1 EOR
%   B3:1/10  "Lock cradle dowm" %
%   N7:1  "Fault Messages" %
% Rung: 147 %
% Cradle Timed Out %
SOR XIC B3:1/15 MOV 10 N7:1 EOR
%   B3:1/15  CRADLE_TIME_OUT  "Cradle movement Time Out" %
%   N7:1  "Fault Messages" %

